C05475=1142.030,341.719,-79.384,-176.572,9.195,148.861
C05476=1142.034,341.471,-79.350,-176.575,9.190,148.861
C05477=1142.038,341.224,-79.316,-176.577,9.187,148.861
C05478=1142.042,340.976,-79.282,-176.580,9.183,148.861
C05479=1142.046,340.728,-79.248,-176.582,9.179,148.860
C05480=1142.050,340.481,-79.214,-176.585,9.175,148.860
C05481=1142.053,340.233,-79.180,-176.588,9.171,148.860
C05482=1142.058,339.985,-79.146,-176.590,9.168,148.859
C05483=1142.062,339.738,-79.112,-176.593,9.164,148.859
C05484=1142.066,339.457,-79.073,-176.595,9.160,148.859
C05485=1142.071,339.176,-79.035,-176.598,9.155,148.858
C05486=1142.075,338.896,-78.997,-176.601,9.150,148.858
C05487=1142.080,338.615,-78.959,-176.604,9.146,148.858
C05488=1142.084,338.368,-78.925,-176.606,9.143,148.857
C05489=1142.088,338.120,-78.891,-176.609,9.139,148.857
C05490=1142.092,337.872,-78.857,-176.612,9.134,148.857
C05491=1142.096,337.625,-78.824,-176.614,9.131,148.857
C05492=1142.100,337.377,-78.790,-176.617,9.127,148.856
C05493=1142.105,337.130,-78.756,-176.619,9.124,148.856
C05494=1142.108,336.881,-78.722,-176.622,9.119,148.856
C05495=1142.112,336.634,-78.689,-176.624,9.116,148.855
C05496=1142.116,336.386,-78.655,-176.627,9.112,148.855
C05497=1142.120,336.139,-78.622,-176.630,9.108,148.855
C05498=1142.124,335.892,-78.588,-176.632,9.104,148.855
C05499=1142.128,335.643,-78.554,-176.635,9.100,148.854
C05500=1142.132,335.395,-78.521,-176.637,9.097,148.854
C05501=1142.136,335.148,-78.487,-176.640,9.093,148.854
C05502=1142.140,334.900,-78.454,-176.642,9.089,148.854
C05503=1142.145,334.653,-78.421,-176.645,9.085,148.853
C05504=1142.148,334.405,-78.387,-176.647,9.082,148.853
C05505=1142.152,334.157,-78.354,-176.650,9.078,148.853
C05506=1142.156,333.909,-78.320,-176.653,9.074,148.853
C05507=1142.161,333.661,-78.287,-176.655,9.070,148.852
C05508=1142.165,333.414,-78.253,-176.658,9.066,148.852
C05509=1142.169,333.166,-78.220,-176.660,9.063,148.852
C05510=1142.172,332.918,-78.186,-176.663,9.059,148.851
C05511=1142.177,332.670,-78.153,-176.666,9.055,148.851
C05512=1142.181,332.422,-78.120,-176.668,9.051,148.851
C05513=1142.185,332.175,-78.086,-176.670,9.048,148.851
C05514=1142.189,331.928,-78.053,-176.673,9.044,148.850
C05515=1142.193,331.680,-78.020,-176.676,9.040,148.850
C05516=1142.197,331.432,-77.986,-176.679,9.036,148.850
C05517=1142.201,331.184,-77.953,-176.681,9.032,148.850
C05518=1142.205,330.936,-77.920,-176.683,9.029,148.849
C05519=1142.209,330.688,-77.887,-176.686,9.025,148.849
C05520=1142.213,330.441,-77.853,-176.689,9.021,148.849
C05521=1142.217,330.193,-77.820,-176.692,9.017,148.849
C05522=1142.221,329.945,-77.787,-176.694,9.014,148.848
C05523=1142.225,329.697,-77.754,-176.697,9.010,148.848
C05524=1142.229,329.450,-77.721,-176.699,9.006,148.848
C05525=1142.234,329.202,-77.688,-176.702,9.002,148.848
C05526=1142.237,328.954,-77.655,-176.704,8.999,148.847
C05527=1142.241,328.707,-77.622,-176.707,8.995,148.847
C05528=1142.245,328.459,-77.589,-176.709,8.992,148.847
C05529=1142.249,328.211,-77.556,-176.712,8.988,148.847
C05530=1142.254,327.964,-77.522,-176.715,8.984,148.847
C05531=1142.258,327.716,-77.489,-176.717,8.980,148.846
C05532=1142.262,327.468,-77.456,-176.719,8.977,148.846
C05533=1142.266,327.220,-77.424,-176.722,8.973,148.846
C05534=1142.270,326.972,-77.391,-176.725,8.969,148.846
C05535=1142.274,326.725,-77.358,-176.728,8.965,148.845
C05536=1142.278,326.477,-77.325,-176.730,8.962,148.845
C05537=1142.282,326.229,-77.292,-176.733,8.958,148.845
C05538=1142.286,325.981,-77.259,-176.735,8.955,148.845
C05539=1142.291,325.733,-77.226,-176.738,8.951,148.844
C05540=1142.294,325.486,-77.194,-176.740,8.947,148.844
C05541=1142.298,325.238,-77.160,-176.743,8.943,148.844
C05542=1142.302,324.990,-77.127,-176.745,8.940,148.844
C05543=1142.307,324.742,-77.095,-176.748,8.936,148.843
C05544=1142.310,324.494,-77.062,-176.750,8.932,148.843
C05545=1142.314,324.247,-77.029,-176.753,8.928,148.843
C05546=1142.319,323.998,-76.997,-176.756,8.925,148.843
C05547=1142.323,323.751,-76.963,-176.759,8.921,148.843
C05548=1142.326,323.503,-76.931,-176.761,8.918,148.842
C05549=1142.331,323.255,-76.898,-176.764,8.914,148.842
C05550=1142.335,323.007,-76.865,-176.766,8.910,148.842
C05551=1142.339,322.759,-76.833,-176.769,8.906,148.842
C05552=1142.343,322.511,-76.800,-176.771,8.903,148.842
C05553=1142.347,322.264,-76.767,-176.774,8.899,148.841
C05554=1142.351,322.016,-76.735,-176.777,8.896,148.841
C05555=1142.355,321.768,-76.702,-176.780,8.892,148.841
C05556=1142.360,321.520,-76.670,-176.782,8.888,148.841
C05557=1142.363,321.273,-76.637,-176.785,8.884,148.840
C05558=1142.368,321.024,-76.605,-176.787,8.881,148.840
C05559=1142.371,320.777,-76.572,-176.790,8.877,148.840
C05560=1142.375,320.529,-76.540,-176.793,8.874,148.840
C05561=1142.380,320.281,-76.507,-176.795,8.870,148.840
C05562=1142.383,320.033,-76.475,-176.798,8.866,148.839
C05563=1142.388,319.785,-76.443,-176.800,8.863,148.839
C05564=1142.392,319.538,-76.410,-176.803,8.859,148.839
C05565=1142.396,319.289,-76.378,-176.805,8.856,148.839
C05566=1142.400,319.042,-76.345,-176.808,8.852,148.839
C05567=1142.404,318.794,-76.313,-176.811,8.848,148.838
C05568=1142.408,318.546,-76.281,-176.814,8.844,148.838
C05569=1142.412,318.298,-76.248,-176.816,8.841,148.838
C05570=1142.416,318.051,-76.216,-176.819,8.837,148.838
C05571=1142.421,317.802,-76.184,-176.821,8.834,148.838
C05572=1142.424,317.555,-76.151,-176.823,8.830,148.837
C05573=1142.428,317.306,-76.119,-176.826,8.826,148.837
C05574=1142.432,317.058,-76.087,-176.829,8.823,148.837
C05575=1142.437,316.811,-76.055,-176.832,8.819,148.837
C05576=1142.441,316.563,-76.023,-176.834,8.816,148.837
C05577=1142.445,316.315,-75.990,-176.837,8.812,148.836
C05578=1142.449,316.067,-75.958,-176.839,8.808,148.836
C05579=1142.453,315.819,-75.926,-176.843,8.805,148.836
C05580=1142.458,315.571,-75.894,-176.845,8.801,148.836
C05581=1142.461,315.323,-75.863,-176.847,8.798,148.836
C05582=1142.465,315.076,-75.829,-176.850,8.794,148.836
C05583=1142.469,314.828,-75.798,-176.853,8.791,148.835
C05584=1142.474,314.580,-75.765,-176.855,8.787,148.835
C05585=1142.478,314.332,-75.734,-176.858,8.783,148.835
C05586=1142.482,314.084,-75.702,-176.860,8.780,148.835
C05587=1142.486,313.835,-75.669,-176.863,8.776,148.835
C05588=1142.490,313.558,-75.634,-176.866,8.772,148.834
C05589=1142.495,313.280,-75.598,-176.869,8.768,148.834
C05590=1142.500,313.003,-75.562,-176.872,8.764,148.834
C05591=1142.504,312.725,-75.526,-176.875,8.760,148.834
C05592=1142.508,312.477,-75.494,-176.878,8.757,148.834
C05593=1142.513,312.229,-75.462,-176.880,8.754,148.833
C05594=1142.516,311.981,-75.431,-176.883,8.750,148.833
C05595=1142.521,311.732,-75.399,-176.885,8.746,148.833
C05596=1142.526,311.485,-75.367,-176.888,8.743,148.833
C05597=1142.529,311.237,-75.335,-176.891,8.739,148.833
C05598=1142.533,310.989,-75.304,-176.893,8.736,148.833
C05599=1142.538,310.741,-75.272,-176.896,8.732,148.832
C05600=1142.542,310.493,-75.240,-176.898,8.729,148.832
C05601=1142.545,310.245,-75.208,-176.901,8.725,148.832
C05602=1142.550,309.998,-75.176,-176.904,8.722,148.832
C05603=1142.553,309.750,-75.145,-176.906,8.718,148.832
C05604=1142.559,309.502,-75.113,-176.909,8.714,148.832
C05605=1142.562,309.253,-75.081,-176.912,8.711,148.832
C05606=1142.566,309.005,-75.049,-176.915,8.707,148.831
C05607=1142.570,308.758,-75.018,-176.917,8.704,148.831
C05608=1142.574,308.509,-74.987,-176.920,8.701,148.831
C05609=1142.580,308.262,-74.955,-176.923,8.697,148.831
C05610=1142.583,308.014,-74.923,-176.925,8.693,148.831
C05611=1142.587,307.766,-74.891,-176.927,8.690,148.831
C05612=1142.592,307.518,-74.860,-176.930,8.686,148.830
C05613=1142.595,307.270,-74.829,-176.933,8.683,148.830
C05614=1142.600,307.022,-74.797,-176.936,8.679,148.830
C05615=1142.604,306.774,-74.766,-176.938,8.676,148.830
C05616=1142.608,306.526,-74.734,-176.941,8.673,148.830
C05617=1142.612,306.278,-74.702,-176.944,8.669,148.830
C05618=1142.617,306.030,-74.671,-176.946,8.666,148.830
C05619=1142.621,305.782,-74.639,-176.949,8.662,148.829
C05620=1142.625,305.533,-74.608,-176.952,8.658,148.829
C05621=1142.629,305.286,-74.577,-176.954,8.655,148.829
C05622=1142.633,305.038,-74.545,-176.957,8.651,148.829
C05623=1142.637,304.790,-74.514,-176.960,8.648,148.829
C05624=1142.641,304.542,-74.482,-176.962,8.645,148.829
C05625=1142.646,304.294,-74.452,-176.965,8.641,148.829
C05626=1142.649,304.046,-74.420,-176.968,8.638,148.829
C05627=1142.654,303.798,-74.389,-176.970,8.634,148.828
C05628=1142.658,303.550,-74.357,-176.973,8.630,148.828
C05629=1142.662,303.302,-74.326,-176.976,8.627,148.828
C05630=1142.667,303.054,-74.296,-176.978,8.624,148.828
C05631=1142.671,302.806,-74.264,-176.981,8.620,148.828
C05632=1142.675,302.558,-74.233,-176.983,8.617,148.828
C05633=1142.679,302.310,-74.201,-176.986,8.614,148.828
C05634=1142.683,302.062,-74.170,-176.989,8.610,148.827
C05635=1142.688,301.813,-74.139,-176.991,8.606,148.827
C05636=1142.692,301.566,-74.108,-176.994,8.604,148.827
C05637=1142.696,301.317,-74.077,-176.997,8.599,148.827
C05638=1142.700,301.070,-74.046,-176.999,8.596,148.827
C05639=1142.704,300.822,-74.015,-177.002,8.593,148.827
C05640=1142.708,300.574,-73.984,-177.005,8.589,148.827
C05641=1142.713,300.326,-73.953,-177.007,8.586,148.827
C05642=1142.716,300.078,-73.921,-177.010,8.583,148.827
C05643=1142.721,299.830,-73.890,-177.013,8.579,148.826
C05644=1142.725,299.581,-73.859,-177.015,8.576,148.826
C05645=1142.729,299.334,-73.829,-177.018,8.573,148.826
C05646=1142.733,299.086,-73.798,-177.021,8.569,148.826
C05647=1142.737,298.838,-73.767,-177.023,8.565,148.826
C05648=1142.742,298.590,-73.736,-177.026,8.562,148.826
C05649=1142.746,298.342,-73.705,-177.029,8.559,148.826
C05650=1142.750,298.093,-73.674,-177.031,8.555,148.825
C05651=1142.754,297.845,-73.644,-177.034,8.552,148.825
C05652=1142.758,297.597,-73.613,-177.037,8.549,148.825
C05653=1142.763,297.349,-73.581,-177.039,8.545,148.825
C05654=1142.767,297.101,-73.550,-177.042,8.542,148.825
C05655=1142.770,296.853,-73.520,-177.045,8.539,148.825
C05656=1142.775,296.605,-73.489,-177.048,8.535,148.825
C05657=1142.780,296.357,-73.458,-177.050,8.532,148.825
C05658=1142.783,296.109,-73.428,-177.053,8.528,148.825
C05659=1142.788,295.861,-73.397,-177.056,8.525,148.825
C05660=1142.792,295.613,-73.366,-177.058,8.521,148.824
C05661=1142.795,295.364,-73.336,-177.061,8.518,148.824
C05662=1142.800,295.117,-73.305,-177.063,8.515,148.824
C05663=1142.805,294.869,-73.274,-177.066,8.511,148.824
C05664=1142.809,294.621,-73.244,-177.069,8.508,148.824
C05665=1142.813,294.372,-73.213,-177.071,8.505,148.824
C05666=1142.817,294.124,-73.182,-177.074,8.501,148.824
C05667=1142.821,293.877,-73.152,-177.077,8.498,148.824
C05668=1142.825,293.628,-73.121,-177.080,8.495,148.824
C05669=1142.830,293.379,-73.091,-177.082,8.492,148.824
C05670=1142.834,293.132,-73.061,-177.085,8.488,148.823
C05671=1142.839,292.884,-73.030,-177.088,8.485,148.823
C05672=1142.842,292.635,-72.999,-177.090,8.481,148.823
C05673=1142.846,292.388,-72.969,-177.093,8.478,148.823
C05674=1142.850,292.140,-72.938,-177.096,8.474,148.823
C05675=1142.855,291.891,-72.908,-177.098,8.471,148.823
C05676=1142.858,291.643,-72.878,-177.101,8.468,148.823
C05677=1142.863,291.395,-72.847,-177.104,8.464,148.823
C05678=1142.868,291.147,-72.816,-177.107,8.461,148.823
C05679=1142.872,290.899,-72.786,-177.109,8.458,148.823
C05680=1142.876,290.651,-72.756,-177.112,8.455,148.823
C05681=1142.880,290.402,-72.725,-177.115,8.451,148.823
C05682=1142.884,290.154,-72.695,-177.118,8.448,148.823
C05683=1142.889,289.906,-72.665,-177.120,8.445,148.822
C05684=1142.893,289.658,-72.634,-177.123,8.442,148.822
C05685=1142.897,289.411,-72.604,-177.126,8.438,148.822
C05686=1142.901,289.162,-72.575,-177.128,8.434,148.822
C05687=1142.905,288.914,-72.544,-177.131,8.432,148.822
C05688=1142.909,288.666,-72.514,-177.133,8.428,148.822
C05689=1142.914,288.417,-72.484,-177.136,8.425,148.822
C05690=1142.918,288.170,-72.453,-177.139,8.421,148.822
C05691=1142.923,287.921,-72.423,-177.142,8.418,148.822
C05692=1142.927,287.646,-72.390,-177.145,8.415,148.822
C05693=1142.932,287.371,-72.356,-177.148,8.410,148.822
C05694=1142.937,287.095,-72.323,-177.151,8.408,148.822
C05695=1142.941,286.820,-72.289,-177.154,8.403,148.821
C05696=1142.945,286.572,-72.260,-177.156,8.401,148.822
C05697=1142.949,286.323,-72.229,-177.159,8.397,148.821
C05698=1142.954,286.075,-72.199,-177.162,8.394,148.821
C05699=1142.957,285.827,-72.169,-177.164,8.390,148.821
C05700=1142.962,285.578,-72.139,-177.167,8.387,148.821
C05701=1142.966,285.331,-72.109,-177.170,8.384,148.821
C05702=1142.970,285.082,-72.080,-177.173,8.380,148.821
C05703=1142.975,284.834,-72.050,-177.175,8.377,148.821
C05704=1142.979,284.586,-72.019,-177.178,8.374,148.821
C05705=1142.983,284.338,-71.990,-177.181,8.371,148.821
C05706=1142.987,284.090,-71.960,-177.183,8.368,148.821
C05707=1142.992,283.842,-71.930,-177.186,8.364,148.821
C05708=1142.996,283.594,-71.900,-177.189,8.361,148.821
C05709=1143.001,283.345,-71.871,-177.192,8.358,148.821
C05710=1143.004,283.098,-71.841,-177.194,8.355,148.821
C05711=1143.009,282.849,-71.811,-177.197,8.352,148.821
C05712=1143.014,282.601,-71.781,-177.200,8.348,148.821
C05713=1143.017,282.353,-71.751,-177.202,8.345,148.820
C05714=1143.022,282.105,-71.721,-177.205,8.342,148.821
C05715=1143.027,281.856,-71.691,-177.208,8.339,148.820
C05716=1143.031,281.608,-71.662,-177.210,8.336,148.820
C05717=1143.035,281.360,-71.633,-177.213,8.332,148.820
C05718=1143.039,281.112,-71.602,-177.216,8.329,148.820
C05719=1143.043,280.864,-71.573,-177.219,8.326,148.820
C05720=1143.047,280.616,-71.543,-177.221,8.322,148.820
C05721=1143.052,280.367,-71.513,-177.224,8.320,148.820
C05722=1143.056,280.119,-71.484,-177.227,8.315,148.820
C05723=1143.060,279.870,-71.454,-177.230,8.313,148.820
C05724=1143.065,279.622,-71.425,-177.232,8.310,148.820
C05725=1143.068,279.375,-71.395,-177.235,8.306,148.820
C05726=1143.073,279.126,-71.365,-177.238,8.303,148.820
C05727=1143.077,278.878,-71.336,-177.241,8.300,148.820
C05728=1143.081,278.630,-71.306,-177.243,8.296,148.820
C05729=1143.085,278.381,-71.277,-177.246,8.293,148.820
C05730=1143.089,278.133,-71.248,-177.248,8.290,148.820
C05731=1143.094,277.885,-71.218,-177.251,8.287,148.820
C05732=1143.098,277.637,-71.189,-177.254,8.284,148.820
C05733=1143.102,277.388,-71.159,-177.257,8.280,148.820
C05734=1143.106,277.140,-71.130,-177.260,8.277,148.820
C05735=1143.111,276.893,-71.101,-177.262,8.274,148.820
C05736=1143.115,276.644,-71.071,-177.265,8.271,148.820
C05737=1143.119,276.396,-71.042,-177.268,8.268,148.820
C05738=1143.124,276.147,-71.013,-177.271,8.264,148.820
C05739=1143.128,275.899,-70.984,-177.273,8.261,148.819
C05740=1143.132,275.651,-70.954,-177.276,8.258,148.820
C05741=1143.136,275.402,-70.925,-177.279,8.255,148.820
C05742=1143.140,275.154,-70.895,-177.281,8.252,148.819
C05743=1143.145,274.906,-70.866,-177.284,8.249,148.819
C05744=1143.149,274.658,-70.837,-177.287,8.246,148.820
C05745=1143.154,274.409,-70.808,-177.290,8.242,148.819
C05746=1143.158,274.161,-70.778,-177.292,8.239,148.819
C05747=1143.162,273.913,-70.749,-177.295,8.236,148.819
C05748=1143.166,273.665,-70.720,-177.298,8.233,148.819
C05749=1143.171,273.416,-70.691,-177.300,8.230,148.819
C05750=1143.176,273.168,-70.662,-177.303,8.227,148.819
C05751=1143.179,272.920,-70.633,-177.306,8.223,148.819
C05752=1143.183,272.672,-70.603,-177.309,8.220,148.819
C05753=1143.188,272.423,-70.575,-177.312,8.217,148.819
C05754=1143.192,272.175,-70.545,-177.314,8.214,148.819
C05755=1143.197,271.927,-70.516,-177.317,8.211,148.819
C05756=1143.201,271.678,-70.487,-177.319,8.208,148.819
C05757=1143.205,271.430,-70.459,-177.322,8.205,148.819
C05758=1143.209,271.182,-70.429,-177.325,8.202,148.819
C05759=1143.214,270.934,-70.401,-177.328,8.198,148.819
C05760=1143.218,270.686,-70.371,-177.331,8.195,148.819
C05761=1143.223,270.437,-70.343,-177.334,8.192,148.819
C05762=1143.226,270.189,-70.314,-177.336,8.189,148.819
C05763=1143.231,269.941,-70.285,-177.339,8.186,148.819
C05764=1143.235,269.692,-70.256,-177.341,8.183,148.819
C05765=1143.240,269.444,-70.226,-177.344,8.180,148.819
C05766=1143.243,269.195,-70.198,-177.347,8.177,148.819
C05767=1143.248,268.948,-70.169,-177.350,8.173,148.819
C05768=1143.253,268.699,-70.140,-177.353,8.170,148.819
C05769=1143.257,268.451,-70.111,-177.355,8.167,148.819
C05770=1143.261,268.203,-70.083,-177.358,8.164,148.819
C05771=1143.266,267.954,-70.054,-177.361,8.161,148.819
C05772=1143.270,267.706,-70.025,-177.363,8.158,148.819
C05773=1143.274,267.457,-69.997,-177.366,8.155,148.819
C05774=1143.278,267.210,-69.968,-177.369,8.152,148.819
C05775=1143.283,266.961,-69.939,-177.372,8.148,148.819
C05776=1143.287,266.712,-69.911,-177.375,8.145,148.819
C05777=1143.291,266.464,-69.882,-177.377,8.143,148.819
C05778=1143.296,266.216,-69.853,-177.380,8.139,148.819
C05779=1143.299,265.968,-69.824,-177.383,8.136,148.819
C05780=1143.304,265.719,-69.796,-177.385,8.133,148.819
C05781=1143.308,265.471,-69.768,-177.388,8.130,148.819
C05782=1143.313,265.223,-69.739,-177.390,8.127,148.819
C05783=1143.317,264.974,-69.710,-177.393,8.124,148.819
C05784=1143.321,264.726,-69.682,-177.396,8.121,148.819
C05785=1143.326,264.478,-69.653,-177.399,8.118,148.819
C05786=1143.330,264.229,-69.625,-177.402,8.115,148.819
C05787=1143.335,263.982,-69.596,-177.405,8.111,148.819
C05788=1143.339,263.733,-69.568,-177.407,8.109,148.819
C05789=1143.343,263.484,-69.539,-177.410,8.106,148.819
C05790=1143.347,263.236,-69.511,-177.413,8.103,148.819
C05791=1143.352,262.987,-69.483,-177.416,8.100,148.819
C05792=1143.357,262.740,-69.454,-177.418,8.096,148.819
C05793=1143.360,262.491,-69.426,-177.421,8.094,148.819
C05794=1143.364,262.243,-69.397,-177.424,8.091,148.819
C05795=1143.369,261.994,-69.369,-177.426,8.088,148.819
C05796=1143.374,261.721,-69.338,-177.430,8.084,148.820
C05797=1143.379,261.447,-69.307,-177.433,8.081,148.820
C05798=1143.383,261.174,-69.275,-177.436,8.077,148.820
C05799=1143.388,260.900,-69.244,-177.439,8.074,148.820
C05800=1143.392,260.652,-69.216,-177.441,8.071,148.820
C05801=1143.397,260.404,-69.188,-177.444,8.068,148.820
C05802=1143.401,260.155,-69.159,-177.447,8.065,148.820
C05803=1143.405,259.907,-69.132,-177.449,8.062,148.820
C05804=1143.410,259.658,-69.103,-177.453,8.059,148.820
C05805=1143.414,259.410,-69.075,-177.456,8.056,148.820
C05806=1143.418,259.162,-69.047,-177.458,8.053,148.820
C05807=1143.423,258.914,-69.019,-177.461,8.049,148.820
C05808=1143.427,258.665,-68.990,-177.463,8.047,148.820
C05809=1143.431,258.417,-68.963,-177.466,8.044,148.820
C05810=1143.436,258.168,-68.934,-177.469,8.041,148.820
C05811=1143.440,257.920,-68.907,-177.472,8.038,148.820
C05812=1143.444,257.671,-68.879,-177.475,8.035,148.820
C05813=1143.449,257.423,-68.850,-177.477,8.032,148.820
C05814=1143.453,257.174,-68.822,-177.480,8.029,148.820
C05815=1143.457,256.927,-68.794,-177.483,8.026,148.820
C05816=1143.462,256.678,-68.766,-177.485,8.023,148.820
C05817=1143.466,256.429,-68.739,-177.488,8.020,148.820
C05818=1143.471,256.181,-68.711,-177.491,8.017,148.820
C05819=1143.474,255.933,-68.683,-177.494,8.014,148.820
C05820=1143.480,255.685,-68.654,-177.497,8.011,148.820
C05821=1143.483,255.436,-68.626,-177.499,8.008,148.820
C05822=1143.488,255.187,-68.599,-177.502,8.005,148.820
C05823=1143.492,254.940,-68.571,-177.504,8.002,148.820
C05824=1143.497,254.691,-68.543,-177.507,7.999,148.820
C05825=1143.501,254.442,-68.516,-177.510,7.996,148.820
C05826=1143.505,254.194,-68.487,-177.513,7.993,148.821
C05827=1143.510,253.946,-68.460,-177.516,7.990,148.821
C05828=1143.514,253.697,-68.433,-177.518,7.987,148.821
C05829=1143.519,253.448,-68.404,-177.522,7.984,148.821
C05830=1143.523,253.200,-68.376,-177.525,7.981,148.821
C05831=1143.527,252.951,-68.349,-177.527,7.978,148.821
C05832=1143.531,252.703,-68.321,-177.530,7.975,148.821
C05833=1143.536,252.455,-68.294,-177.533,7.972,148.821
C05834=1143.540,252.206,-68.266,-177.535,7.969,148.821
C05835=1143.544,251.958,-68.238,-177.538,7.966,148.821
C05836=1143.550,251.710,-68.210,-177.541,7.963,148.821
C05837=1143.553,251.461,-68.182,-177.544,7.960,148.821
C05838=1143.558,251.213,-68.155,-177.546,7.957,148.821
C05839=1143.562,250.965,-68.127,-177.549,7.954,148.821
C05840=1143.566,250.716,-68.100,-177.552,7.951,148.821
C05841=1143.571,250.468,-68.072,-177.555,7.948,148.821
C05842=1143.575,250.219,-68.045,-177.558,7.945,148.821
C05843=1143.579,249.971,-68.017,-177.560,7.942,148.821
C05844=1143.584,249.722,-67.990,-177.563,7.939,148.822
C05845=1143.589,249.474,-67.963,-177.566,7.937,148.822
C05846=1143.593,249.226,-67.935,-177.569,7.934,148.822
C05847=1143.597,248.976,-67.907,-177.572,7.931,148.822
C05848=1143.601,248.729,-67.880,-177.574,7.928,148.822
C05849=1143.606,248.480,-67.853,-177.577,7.925,148.822
C05850=1143.610,248.231,-67.825,-177.580,7.922,148.822
C05851=1143.614,247.983,-67.797,-177.583,7.919,148.822
C05852=1143.619,247.735,-67.770,-177.585,7.917,148.822
C05853=1143.624,247.486,-67.743,-177.588,7.914,148.822
C05854=1143.627,247.237,-67.715,-177.590,7.911,148.822
C05855=1143.632,246.989,-67.688,-177.593,7.908,148.822
C05856=1143.637,246.740,-67.661,-177.596,7.905,148.822
C05857=1143.641,246.492,-67.634,-177.599,7.902,148.823
C05858=1143.646,246.244,-67.606,-177.601,7.899,148.822
C05859=1143.650,245.995,-67.579,-177.604,7.896,148.822
C05860=1143.654,245.746,-67.552,-177.607,7.893,148.823
C05861=1143.658,245.498,-67.525,-177.610,7.890,148.823
C05862=1143.663,245.250,-67.497,-177.612,7.887,148.823
C05863=1143.667,245.002,-67.470,-177.615,7.884,148.823
C05864=1143.671,244.753,-67.443,-177.618,7.882,148.823
C05865=1143.676,244.504,-67.416,-177.621,7.879,148.823
C05866=1143.681,244.256,-67.389,-177.624,7.876,148.823
C05867=1143.685,244.007,-67.362,-177.626,7.873,148.823
C05868=1143.689,243.759,-67.335,-177.630,7.870,148.823
C05869=1143.693,243.510,-67.307,-177.632,7.867,148.823
C05870=1143.698,243.262,-67.280,-177.635,7.864,148.824
C05871=1143.702,243.013,-67.253,-177.638,7.861,148.824
C05872=1143.707,242.765,-67.226,-177.641,7.858,148.824
C05873=1143.711,242.517,-67.200,-177.644,7.856,148.824
C05874=1143.716,242.268,-67.172,-177.646,7.853,148.824
C05875=1143.720,242.020,-67.145,-177.649,7.850,148.824
C05876=1143.724,241.771,-67.118,-177.652,7.847,148.824
C05877=1143.728,241.522,-67.092,-177.654,7.845,148.824
C05878=1143.733,241.274,-67.064,-177.657,7.842,148.824
C05879=1143.738,241.025,-67.037,-177.660,7.839,148.824
C05880=1143.742,240.777,-67.010,-177.662,7.836,148.824
C05881=1143.746,240.529,-66.984,-177.665,7.833,148.824
C05882=1143.751,240.280,-66.957,-177.668,7.830,148.824
C05883=1143.755,240.032,-66.930,-177.671,7.827,148.825
C05884=1143.760,239.783,-66.904,-177.674,7.824,148.825
C05885=1143.764,239.534,-66.877,-177.676,7.821,148.825
C05886=1143.769,239.286,-66.850,-177.679,7.818,148.825
C05887=1143.772,239.037,-66.823,-177.682,7.816,148.825
C05888=1143.777,238.789,-66.796,-177.685,7.813,148.825
C05889=1143.782,238.540,-66.769,-177.688,7.810,148.825
C05890=1143.786,238.292,-66.742,-177.690,7.807,148.825
C05891=1143.790,238.043,-66.716,-177.693,7.805,148.825
C05892=1143.795,237.794,-66.689,-177.695,7.802,148.825
C05893=1143.799,237.546,-66.663,-177.699,7.799,148.826
C05894=1143.804,237.298,-66.636,-177.701,7.796,148.826
C05895=1143.808,237.049,-66.610,-177.704,7.793,148.826
C05896=1143.813,236.800,-66.583,-177.707,7.790,148.826
C05897=1143.817,236.552,-66.556,-177.710,7.787,148.826
C05898=1143.821,236.304,-66.529,-177.713,7.785,148.826
C05899=1143.826,236.054,-66.503,-177.715,7.782,148.826
C05900=1143.831,235.783,-66.474,-177.718,7.779,148.826
C05901=1143.836,235.512,-66.445,-177.721,7.776,148.826
C05902=1143.840,235.239,-66.416,-177.724,7.773,148.827
C05903=1143.845,234.967,-66.387,-177.728,7.769,148.827
C05904=1143.850,234.719,-66.360,-177.730,7.767,148.827
C05905=1143.854,234.470,-66.334,-177.733,7.764,148.827
C05906=1143.858,234.222,-66.307,-177.735,7.762,148.827
C05907=1143.863,233.973,-66.281,-177.738,7.759,148.827
C05908=1143.867,233.724,-66.254,-177.741,7.756,148.827
C05909=1143.871,233.476,-66.228,-177.744,7.753,148.827
C05910=1143.876,233.227,-66.201,-177.747,7.750,148.827
C05911=1143.881,232.980,-66.175,-177.750,7.747,148.828
C05912=1143.886,232.730,-66.149,-177.753,7.744,148.828
C05913=1143.890,232.482,-66.123,-177.755,7.741,148.828
C05914=1143.895,232.233,-66.096,-177.758,7.739,148.828
C05915=1143.898,231.985,-66.070,-177.761,7.736,148.828
C05916=1143.903,231.736,-66.044,-177.763,7.734,148.828
C05917=1143.907,231.488,-66.017,-177.766,7.731,148.828
C05918=1143.912,231.239,-65.991,-177.769,7.728,148.828
C05919=1143.917,230.990,-65.965,-177.772,7.725,148.828
C05920=1143.920,230.742,-65.938,-177.775,7.722,148.829
C05921=1143.925,230.493,-65.913,-177.778,7.719,148.829
C05922=1143.930,230.245,-65.886,-177.780,7.717,148.829
C05923=1143.934,229.996,-65.860,-177.783,7.714,148.829
C05924=1143.938,229.747,-65.834,-177.786,7.711,148.829
C05925=1143.943,229.499,-65.807,-177.788,7.708,148.829
C05926=1143.947,229.250,-65.782,-177.792,7.706,148.829
C05927=1143.951,229.001,-65.756,-177.794,7.703,148.829
C05928=1143.957,228.753,-65.729,-177.797,7.701,148.829
C05929=1143.961,228.505,-65.703,-177.799,7.698,148.830
C05930=1143.965,228.256,-65.678,-177.802,7.695,148.830
C05931=1143.969,228.007,-65.652,-177.805,7.692,148.830
C05932=1143.974,227.758,-65.625,-177.808,7.690,148.830
C05933=1143.978,227.510,-65.599,-177.811,7.687,148.830
C05934=1143.983,227.262,-65.574,-177.814,7.684,148.830
C05935=1143.987,227.013,-65.548,-177.816,7.682,148.830
C05936=1143.992,226.764,-65.521,-177.819,7.679,148.830
C05937=1143.996,226.515,-65.495,-177.822,7.676,148.831
C05938=1144.000,226.267,-65.469,-177.825,7.673,148.831
C05939=1144.005,226.019,-65.444,-177.828,7.670,148.831
C05940=1144.010,225.769,-65.418,-177.831,7.667,148.831
C05941=1144.014,225.521,-65.392,-177.833,7.665,148.831
C05942=1144.019,225.272,-65.366,-177.836,7.662,148.831
C05943=1144.023,225.024,-65.340,-177.839,7.660,148.832
C05944=1144.027,224.776,-65.314,-177.842,7.657,148.832
C05945=1144.032,224.527,-65.289,-177.844,7.654,148.832
C05946=1144.037,224.278,-65.262,-177.847,7.652,148.832
C05947=1144.041,224.030,-65.237,-177.849,7.649,148.832
C05948=1144.046,223.781,-65.211,-177.853,7.646,148.832
C05949=1144.050,223.532,-65.185,-177.855,7.643,148.832
C05950=1144.054,223.283,-65.160,-177.858,7.641,148.832
C05951=1144.059,223.035,-65.134,-177.860,7.638,148.833
C05952=1144.063,222.786,-65.108,-177.863,7.636,148.833
C05953=1144.067,222.537,-65.083,-177.867,7.633,148.833
C05954=1144.072,222.289,-65.057,-177.869,7.630,148.833
C05955=1144.076,222.040,-65.032,-177.872,7.627,148.833
C05956=1144.081,221.791,-65.005,-177.874,7.625,148.833
C05957=1144.086,221.543,-64.980,-177.877,7.622,148.833
C05958=1144.090,221.294,-64.954,-177.880,7.620,148.834
C05959=1144.095,221.045,-64.929,-177.883,7.617,148.834
C05960=1144.100,220.797,-64.904,-177.886,7.614,148.834
C05961=1144.104,220.548,-64.878,-177.888,7.612,148.834
C05962=1144.108,220.299,-64.852,-177.891,7.609,148.834
C05963=1144.113,220.051,-64.827,-177.894,7.606,148.834
C05964=1144.117,219.802,-64.801,-177.897,7.603,148.834
C05965=1144.122,219.554,-64.775,-177.900,7.600,148.835
C05966=1144.127,219.305,-64.751,-177.903,7.599,148.835
C05967=1144.131,219.056,-64.725,-177.905,7.596,148.835
C05968=1144.135,218.807,-64.699,-177.908,7.593,148.835
C05969=1144.139,218.560,-64.674,-177.911,7.590,148.835
C05970=1144.143,218.311,-64.649,-177.914,7.588,148.835
C05971=1144.149,218.062,-64.624,-177.916,7.585,148.836
C05972=1144.153,217.813,-64.598,-177.919,7.582,148.836
C05973=1144.157,217.564,-64.572,-177.922,7.579,148.836
C05974=1144.162,217.316,-64.548,-177.925,7.578,148.836
C05975=1144.166,217.067,-64.522,-177.927,7.575,148.836
C05976=1144.171,216.819,-64.497,-177.930,7.572,148.836
C05977=1144.176,216.569,-64.472,-177.933,7.569,148.836
C05978=1144.180,216.320,-64.446,-177.936,7.566,148.837
C05979=1144.184,216.073,-64.421,-177.939,7.564,148.837
C05980=1144.189,215.823,-64.396,-177.941,7.561,148.837
C05981=1144.193,215.575,-64.371,-177.945,7.559,148.837
C05982=1144.198,215.326,-64.345,-177.947,7.556,148.837
C05983=1144.203,215.078,-64.320,-177.950,7.554,148.837
C05984=1144.207,214.829,-64.294,-177.952,7.551,148.838
C05985=1144.211,214.580,-64.270,-177.956,7.548,148.838
C05986=1144.216,214.332,-64.245,-177.958,7.546,148.838
C05987=1144.220,214.082,-64.220,-177.961,7.543,148.838
C05988=1144.225,213.834,-64.194,-177.964,7.541,148.838
C05989=1144.229,213.585,-64.169,-177.967,7.538,148.839
C05990=1144.234,213.337,-64.144,-177.969,7.536,148.839
C05991=1144.238,213.087,-64.119,-177.972,7.533,148.839
C05992=1144.243,212.839,-64.094,-177.975,7.530,148.839
C05993=1144.247,212.590,-64.069,-177.978,7.527,148.839
C05994=1144.252,212.342,-64.044,-177.980,7.525,148.839
C05995=1144.256,212.093,-64.019,-177.983,7.523,148.840
C05996=1144.261,211.845,-63.994,-177.986,7.520,148.840
C05997=1144.265,211.596,-63.970,-177.988,7.518,148.840
C05998=1144.270,211.347,-63.945,-177.992,7.515,148.840
C05999=1144.275,211.099,-63.919,-177.994,7.512,148.840
C06000=1144.278,210.850,-63.895,-177.997,7.509,148.840
C06001=1144.284,210.601,-63.870,-178.000,7.507,148.841
C06002=1144.288,210.352,-63.844,-178.003,7.505,148.841
C06003=1144.292,210.104,-63.820,-178.006,7.502,148.841
C06004=1144.297,209.832,-63.793,-178.009,7.499,148.841
C06005=1144.303,209.562,-63.766,-178.012,7.496,148.841
C06006=1144.307,209.291,-63.739,-178.015,7.494,148.842
C06007=1144.312,209.021,-63.712,-178.018,7.491,148.842
C06008=1144.317,208.772,-63.687,-178.020,7.489,148.842
C06009=1144.321,208.524,-63.662,-178.023,7.486,148.842
C06010=1144.325,208.275,-63.637,-178.026,7.483,148.842
C06011=1144.330,208.026,-63.613,-178.029,7.481,148.843
C06012=1144.335,207.777,-63.588,-178.031,7.478,148.843
C06013=1144.340,207.528,-63.563,-178.034,7.476,148.843
C06014=1144.344,207.280,-63.539,-178.038,7.473,148.843
C06015=1144.349,207.031,-63.514,-178.040,7.471,148.843
C06016=1144.353,206.782,-63.490,-178.043,7.468,148.843
C06017=1144.358,206.534,-63.465,-178.046,7.465,148.844
C06018=1144.361,206.285,-63.440,-178.048,7.463,148.844
C06019=1144.367,206.036,-63.416,-178.051,7.461,148.844
C06020=1144.371,205.787,-63.392,-178.054,7.458,148.844
C06021=1144.375,205.539,-63.366,-178.056,7.456,148.844
C06022=1144.380,205.290,-63.342,-178.060,7.453,148.845
C06023=1144.385,205.041,-63.317,-178.062,7.450,148.845
C06024=1144.389,204.793,-63.293,-178.065,7.449,148.845
C06025=1144.394,204.544,-63.268,-178.068,7.446,148.845
C06026=1144.398,204.295,-63.244,-178.071,7.443,148.845
C06027=1144.403,204.046,-63.219,-178.073,7.441,148.846
C06028=1144.407,203.797,-63.195,-178.076,7.438,148.846
C06029=1144.412,203.549,-63.170,-178.079,7.435,148.846
C06030=1144.417,203.300,-63.146,-178.082,7.433,148.846
C06031=1144.420,203.051,-63.122,-178.084,7.430,148.846
C06032=1144.425,202.802,-63.097,-178.088,7.428,148.847
C06033=1144.430,202.554,-63.073,-178.090,7.426,148.847
C06034=1144.435,202.305,-63.048,-178.093,7.423,148.847
C06035=1144.439,202.056,-63.025,-178.095,7.421,148.847
C06036=1144.443,201.807,-63.001,-178.098,7.418,148.847
C06037=1144.449,201.558,-62.976,-178.102,7.416,148.848
C06038=1144.452,201.309,-62.951,-178.104,7.414,148.848
C06039=1144.457,201.061,-62.927,-178.107,7.411,148.848
C06040=1144.462,200.812,-62.903,-178.110,7.408,148.848
C06041=1144.466,200.564,-62.879,-178.113,7.406,148.849
C06042=1144.471,200.315,-62.855,-178.115,7.404,148.849
C06043=1144.476,200.065,-62.830,-178.118,7.401,148.849
C06044=1144.480,199.817,-62.806,-178.121,7.399,148.849
C06045=1144.484,199.568,-62.782,-178.124,7.396,148.849
C06046=1144.489,199.320,-62.757,-178.126,7.394,148.850
C06047=1144.494,199.070,-62.734,-178.129,7.391,148.850
C06048=1144.498,198.822,-62.710,-178.132,7.389,148.850
C06049=1144.502,198.573,-62.685,-178.135,7.387,148.850
C06050=1144.507,198.324,-62.661,-178.138,7.384,148.851
C06051=1144.512,198.075,-62.637,-178.140,7.382,148.851
C06052=1144.517,197.827,-62.613,-178.143,7.379,148.851
C06053=1144.520,197.578,-62.589,-178.146,7.377,148.851
C06054=1144.526,197.329,-62.565,-178.148,7.374,148.851
C06055=1144.530,197.080,-62.541,-178.152,7.372,148.852
C06056=1144.535,196.832,-62.517,-178.154,7.370,148.852
C06057=1144.539,196.583,-62.493,-178.157,7.367,148.852
C06058=1144.544,196.334,-62.469,-178.160,7.364,148.852
C06059=1144.548,196.085,-62.444,-178.163,7.363,148.853
C06060=1144.553,195.836,-62.421,-178.165,7.360,148.853
C06061=1144.557,195.587,-62.397,-178.168,7.358,148.853
C06062=1144.562,195.338,-62.374,-178.171,7.355,148.853
C06063=1144.566,195.090,-62.350,-178.174,7.353,148.853
C06064=1144.571,194.841,-62.326,-178.176,7.350,148.854
C06065=1144.576,194.592,-62.301,-178.180,7.348,148.854
C06066=1144.581,194.343,-62.278,-178.182,7.346,148.854
C06067=1144.585,194.095,-62.254,-178.185,7.343,148.854
C06068=1144.589,193.845,-62.230,-178.187,7.341,148.855
C06069=1144.594,193.597,-62.206,-178.191,7.339,148.855
C06070=1144.599,193.348,-62.183,-178.194,7.336,148.855
C06071=1144.603,193.099,-62.159,-178.196,7.334,148.855
C06072=1144.608,192.850,-62.135,-178.199,7.331,148.855
C06073=1144.612,192.602,-62.111,-178.202,7.329,148.856
C06074=1144.617,192.353,-62.088,-178.205,7.326,148.856
C06075=1144.621,192.104,-62.064,-178.207,7.325,148.856
C06076=1144.626,191.855,-62.041,-178.210,7.322,148.856
C06077=1144.631,191.606,-62.017,-178.213,7.319,148.857
C06078=1144.636,191.357,-61.993,-178.216,7.317,148.857
C06079=1144.640,191.108,-61.969,-178.219,7.315,148.857
C06080=1144.645,190.859,-61.946,-178.221,7.312,148.857
C06081=1144.649,190.611,-61.922,-178.224,7.310,148.858
C06082=1144.654,190.362,-61.898,-178.227,7.308,148.858
C06083=1144.659,190.113,-61.875,-178.230,7.305,148.858
C06084=1144.663,189.865,-61.851,-178.233,7.304,148.858
C06085=1144.668,189.616,-61.828,-178.235,7.301,148.859
C06086=1144.672,189.367,-61.805,-178.238,7.299,148.859
C06087=1144.677,189.118,-61.781,-178.241,7.296,148.859
C06088=1144.681,188.869,-61.757,-178.244,7.293,148.859
C06089=1144.686,188.620,-61.734,-178.246,7.291,148.860
C06090=1144.690,188.371,-61.711,-178.250,7.289,148.860
C06091=1144.695,188.122,-61.687,-178.252,7.287,148.860
C06092=1144.699,187.874,-61.663,-178.255,7.284,148.860
C06093=1144.704,187.625,-61.640,-178.258,7.282,148.861
C06094=1144.709,187.376,-61.617,-178.261,7.280,148.861
C06095=1144.714,187.127,-61.593,-178.263,7.278,148.861
C06096=1144.718,186.878,-61.570,-178.266,7.275,148.861
C06097=1144.723,186.629,-61.546,-178.269,7.273,148.862
C06098=1144.727,186.380,-61.524,-178.272,7.270,148.862
C06099=1144.731,186.132,-61.500,-178.274,7.268,148.862
C06100=1144.736,185.882,-61.476,-178.277,7.266,148.862
C06101=1144.741,185.633,-61.453,-178.280,7.264,148.863
C06102=1144.746,185.385,-61.430,-178.283,7.261,148.863
C06103=1144.751,185.136,-61.407,-178.285,7.259,148.863
C06104=1144.755,184.887,-61.384,-178.289,7.257,148.863
C06105=1144.759,184.638,-61.360,-178.291,7.255,148.864
C06106=1144.764,184.389,-61.337,-178.294,7.252,148.864
C06107=1144.769,184.140,-61.314,-178.297,7.250,148.864
C06108=1144.773,183.871,-61.289,-178.300,7.247,148.864
C06109=1144.779,183.601,-61.264,-178.303,7.245,148.865
C06110=1144.784,183.332,-61.239,-178.306,7.242,148.865
C06111=1144.789,183.062,-61.213,-178.308,7.240,148.865
C06112=1144.793,182.813,-61.191,-178.312,7.238,148.866
C06113=1144.798,182.564,-61.167,-178.314,7.236,148.866
C06114=1144.802,182.315,-61.144,-178.317,7.233,148.866
C06115=1144.807,182.066,-61.121,-178.320,7.231,148.866
C06116=1144.811,181.817,-61.099,-178.323,7.229,148.867
C06117=1144.816,181.568,-61.075,-178.325,7.227,148.867
C06118=1144.821,181.320,-61.052,-178.329,7.224,148.867
C06119=1144.825,181.071,-61.029,-178.331,7.222,148.867
C06120=1144.830,180.822,-61.006,-178.334,7.219,148.868
C06121=1144.835,180.573,-60.983,-178.337,7.218,148.868
C06122=1144.839,180.324,-60.960,-178.340,7.215,148.868
C06123=1144.844,180.075,-60.938,-178.342,7.213,148.869
C06124=1144.849,179.826,-60.914,-178.345,7.210,148.869
C06125=1144.853,179.577,-60.892,-178.348,7.208,148.869
C06126=1144.858,179.328,-60.868,-178.351,7.206,148.869
C06127=1144.862,179.079,-60.846,-178.353,7.204,148.870
C06128=1144.867,178.831,-60.823,-178.356,7.202,148.870
C06129=1144.872,178.582,-60.800,-178.359,7.200,148.870
C06130=1144.876,178.333,-60.777,-178.362,7.198,148.870
C06131=1144.881,178.083,-60.754,-178.365,7.195,148.871
C06132=1144.885,177.835,-60.732,-178.368,7.193,148.871
C06133=1144.890,177.586,-60.709,-178.370,7.190,148.871
C06134=1144.894,177.337,-60.687,-178.373,7.189,148.872
C06135=1144.899,177.088,-60.663,-178.376,7.186,148.872
C06136=1144.904,176.840,-60.640,-178.379,7.184,148.872
C06137=1144.909,176.590,-60.618,-178.382,7.181,148.872
C06138=1144.913,176.341,-60.595,-178.385,7.180,148.873
C06139=1144.917,176.092,-60.572,-178.387,7.178,148.873
C06140=1144.923,175.844,-60.550,-178.390,7.175,148.873
C06141=1144.927,175.595,-60.527,-178.393,7.173,148.874
C06142=1144.932,175.345,-60.504,-178.396,7.170,148.874
C06143=1144.936,175.097,-60.482,-178.398,7.169,148.874
C06144=1144.941,174.847,-60.459,-178.402,7.166,148.875
C06145=1144.945,174.599,-60.437,-178.404,7.164,148.875
C06146=1144.951,174.350,-60.414,-178.406,7.162,148.875
C06147=1144.955,174.101,-60.392,-178.410,7.160,148.875
C06148=1144.959,173.852,-60.369,-178.412,7.158,148.876
C06149=1144.965,173.603,-60.347,-178.415,7.155,148.876
C06150=1144.969,173.355,-60.324,-178.418,7.153,148.876
C06151=1144.974,173.105,-60.301,-178.420,7.151,148.876
C06152=1144.978,172.856,-60.279,-178.424,7.149,148.877
C06153=1144.983,172.607,-60.256,-178.426,7.147,148.877
C06154=1144.987,172.358,-60.234,-178.429,7.144,148.877
C06155=1144.992,172.110,-60.212,-178.432,7.142,148.878
C06156=1144.997,171.860,-60.189,-178.434,7.141,148.878
C06157=1145.001,171.612,-60.166,-178.437,7.138,148.878
C06158=1145.006,171.363,-60.145,-178.440,7.136,148.879
C06159=1145.011,171.113,-60.122,-178.443,7.134,148.879
C06160=1145.015,170.865,-60.099,-178.446,7.132,148.879
C06161=1145.020,170.616,-60.077,-178.448,7.130,148.879
C06162=1145.025,170.366,-60.055,-178.451,7.127,148.880
C06163=1145.029,170.118,-60.032,-178.454,7.126,148.880
C06164=1145.034,169.869,-60.010,-178.457,7.123,148.880
C06165=1145.039,169.620,-59.988,-178.460,7.121,148.881
C06166=1145.043,169.371,-59.965,-178.462,7.119,148.881
C06167=1145.047,169.122,-59.943,-178.466,7.117,148.881
C06168=1145.053,168.873,-59.921,-178.468,7.115,148.881
C06169=1145.057,168.624,-59.899,-178.471,7.112,148.882
C06170=1145.062,168.376,-59.877,-178.474,7.110,148.882
C06171=1145.067,168.126,-59.854,-178.476,7.108,148.882
C06172=1145.072,167.877,-59.832,-178.479,7.106,148.883
C06173=1145.076,167.628,-59.810,-178.482,7.104,148.883
C06174=1145.081,167.379,-59.788,-178.485,7.102,148.883
C06175=1145.085,167.130,-59.765,-178.488,7.099,148.884
C06176=1145.090,166.882,-59.743,-178.490,7.098,148.884
C06177=1145.095,166.632,-59.721,-178.493,7.096,148.884
C06178=1145.099,166.384,-59.700,-178.496,7.093,148.885
C06179=1145.104,166.134,-59.678,-178.499,7.091,148.885
C06180=1145.109,165.885,-59.655,-178.502,7.089,148.885
C06181=1145.114,165.636,-59.633,-178.505,7.087,148.886
C06182=1145.118,165.387,-59.612,-178.507,7.085,148.886
C06183=1145.123,165.138,-59.590,-178.510,7.082,148.886
C06184=1145.127,164.890,-59.567,-178.513,7.081,148.886
C06185=1145.132,164.641,-59.545,-178.515,7.079,148.887
C06186=1145.136,164.392,-59.523,-178.519,7.076,148.887
C06187=1145.141,164.142,-59.501,-178.521,7.074,148.887
C06188=1145.146,163.894,-59.479,-178.524,7.073,148.888
C06189=1145.151,163.644,-59.457,-178.527,7.070,148.888
C06190=1145.155,163.396,-59.435,-178.530,7.068,148.888
C06191=1145.160,163.146,-59.413,-178.532,7.066,148.889
C06192=1145.165,162.898,-59.392,-178.535,7.064,148.889
C06193=1145.169,162.648,-59.370,-178.538,7.062,148.889
C06194=1145.174,162.400,-59.348,-178.541,7.060,148.890
C06195=1145.178,162.151,-59.326,-178.544,7.058,148.890
C06196=1145.183,161.901,-59.305,-178.546,7.056,148.890
C06197=1145.188,161.653,-59.283,-178.549,7.054,148.891
C06198=1145.192,161.403,-59.261,-178.552,7.051,148.891
C06199=1145.197,161.155,-59.240,-178.555,7.050,148.891
C06200=1145.201,160.905,-59.217,-178.558,7.048,148.892
C06201=1145.206,160.657,-59.196,-178.560,7.045,148.892
C06202=1145.211,160.408,-59.174,-178.563,7.043,148.892
C06203=1145.215,160.159,-59.152,-178.566,7.042,148.893
C06204=1145.221,159.909,-59.131,-178.568,7.040,148.893
C06205=1145.225,159.660,-59.109,-178.571,7.037,148.893
C06206=1145.230,159.411,-59.087,-178.574,7.035,148.893
C06207=1145.235,159.163,-59.066,-178.577,7.034,148.894
C06208=1145.239,158.913,-59.044,-178.580,7.031,148.894
C06209=1145.244,158.664,-59.023,-178.583,7.029,148.895
C06210=1145.249,158.416,-59.001,-178.585,7.028,148.895
C06211=1145.253,158.166,-58.979,-178.588,7.025,148.895
C06212=1145.259,157.897,-58.956,-178.591,7.023,148.895
C06213=1145.263,157.628,-58.932,-178.594,7.020,148.896
C06214=1145.269,157.359,-58.909,-178.597,7.019,148.896
C06215=1145.273,157.090,-58.886,-178.600,7.016,148.897
C06216=1145.278,156.841,-58.864,-178.603,7.014,148.897
C06217=1145.283,156.593,-58.843,-178.606,7.013,148.897
C06218=1145.288,156.343,-58.822,-178.609,7.010,148.898
C06219=1145.293,156.094,-58.800,-178.611,7.008,148.898
C06220=1145.298,155.845,-58.779,-178.614,7.006,148.898
C06221=1145.303,155.596,-58.757,-178.617,7.005,148.899
C06222=1145.306,155.347,-58.736,-178.620,7.002,148.899
C06223=1145.311,155.098,-58.715,-178.623,7.000,148.899
C06224=1145.316,154.849,-58.693,-178.625,6.999,148.900
C06225=1145.321,154.600,-58.672,-178.628,6.996,148.900
C06226=1145.326,154.351,-58.650,-178.631,6.994,148.900
C06227=1145.330,154.102,-58.628,-178.634,6.992,148.901
C06228=1145.335,153.853,-58.608,-178.636,6.991,148.901
C06229=1145.339,153.604,-58.586,-178.640,6.988,148.901
C06230=1145.344,153.354,-58.565,-178.642,6.986,148.902
C06231=1145.349,153.106,-58.543,-178.645,6.985,148.902
C06232=1145.354,152.857,-58.523,-178.647,6.983,148.902
C06233=1145.359,152.608,-58.501,-178.650,6.980,148.903
C06234=1145.363,152.358,-58.480,-178.653,6.978,148.903
C06235=1145.368,152.110,-58.458,-178.656,6.977,148.903
C06236=1145.372,151.861,-58.438,-178.659,6.975,148.904
C06237=1145.378,151.611,-58.417,-178.662,6.972,148.904
C06238=1145.382,151.362,-58.395,-178.665,6.971,148.905
C06239=1145.387,151.113,-58.374,-178.667,6.969,148.905
C06240=1145.391,150.865,-58.353,-178.670,6.967,148.905
C06241=1145.396,150.615,-58.332,-178.673,6.964,148.905
C06242=1145.402,150.366,-58.311,-178.676,6.963,148.906
C06243=1145.406,150.118,-58.290,-178.678,6.961,148.906
C06244=1145.410,149.868,-58.268,-178.681,6.959,148.907
C06245=1145.415,149.618,-58.247,-178.684,6.958,148.907
C06246=1145.420,149.370,-58.226,-178.686,6.955,148.907
C06247=1145.425,149.121,-58.205,-178.689,6.953,148.908
C06248=1145.430,148.872,-58.184,-178.692,6.951,148.908
C06249=1145.434,148.623,-58.163,-178.695,6.950,148.908
C06250=1145.439,148.373,-58.142,-178.698,6.947,148.909
C06251=1145.444,148.124,-58.121,-178.701,6.945,148.909
C06252=1145.448,147.876,-58.100,-178.703,6.944,148.909
C06253=1145.453,147.626,-58.079,-178.706,6.942,148.910
C06254=1145.457,147.378,-58.058,-178.709,6.940,148.910
C06255=1145.463,147.128,-58.037,-178.712,6.937,148.910
C06256=1145.468,146.879,-58.016,-178.714,6.936,148.911
C06257=1145.471,146.630,-57.995,-178.717,6.934,148.911
C06258=1145.477,146.381,-57.974,-178.720,6.932,148.912
C06259=1145.481,146.132,-57.954,-178.722,6.930,148.912
C06260=1145.486,145.882,-57.933,-178.726,6.928,148.912
C06261=1145.491,145.634,-57.912,-178.728,6.926,148.913
C06262=1145.495,145.385,-57.891,-178.731,6.924,148.913
C06263=1145.500,145.136,-57.870,-178.734,6.923,148.913
C06264=1145.505,144.887,-57.849,-178.737,6.921,148.914
C06265=1145.510,144.638,-57.829,-178.739,6.918,148.914
C06266=1145.515,144.388,-57.808,-178.742,6.916,148.914
C06267=1145.519,144.140,-57.788,-178.745,6.915,148.915
C06268=1145.524,143.890,-57.767,-178.748,6.913,148.915
C06269=1145.528,143.641,-57.746,-178.750,6.911,148.916
C06270=1145.533,143.391,-57.725,-178.754,6.909,148.916
C06271=1145.538,143.142,-57.705,-178.756,6.907,148.916
C06272=1145.543,142.893,-57.684,-178.759,6.905,148.917
C06273=1145.547,142.644,-57.663,-178.762,6.904,148.917
C06274=1145.553,142.395,-57.642,-178.764,6.902,148.917
C06275=1145.557,142.146,-57.622,-178.767,6.900,148.918
C06276=1145.561,141.897,-57.602,-178.770,6.898,148.918
C06277=1145.567,141.648,-57.581,-178.773,6.896,148.919
C06278=1145.571,141.399,-57.560,-178.776,6.894,148.919
C06279=1145.576,141.150,-57.539,-178.778,6.892,148.919
C06280=1145.581,140.901,-57.519,-178.781,6.890,148.920
C06281=1145.585,140.652,-57.498,-178.784,6.889,148.920
C06282=1145.590,140.402,-57.478,-178.787,6.886,148.920
C06283=1145.595,140.153,-57.457,-178.790,6.885,148.921
C06284=1145.600,139.904,-57.436,-178.792,6.883,148.921
C06285=1145.604,139.655,-57.416,-178.795,6.881,148.921
C06286=1145.609,139.406,-57.395,-178.798,6.879,148.922
C06287=1145.614,139.156,-57.375,-178.800,6.878,148.922
C06288=1145.619,138.907,-57.355,-178.803,6.876,148.923
C06289=1145.623,138.659,-57.334,-178.806,6.873,148.923
C06290=1145.628,138.409,-57.313,-178.809,6.872,148.923
C06291=1145.633,138.160,-57.293,-178.812,6.870,148.924
C06292=1145.638,137.912,-57.273,-178.815,6.868,148.924
C06293=1145.642,137.663,-57.253,-178.817,6.867,148.925
C06294=1145.648,137.413,-57.232,-178.820,6.865,148.925
C06295=1145.652,137.164,-57.212,-178.823,6.863,148.925
C06296=1145.657,136.915,-57.192,-178.825,6.862,148.926
C06297=1145.661,136.666,-57.172,-178.829,6.859,148.926
C06298=1145.666,136.417,-57.151,-178.831,6.857,148.927
C06299=1145.671,136.168,-57.131,-178.834,6.856,148.927
C06300=1145.675,135.919,-57.110,-178.837,6.854,148.927
C06301=1145.680,135.669,-57.091,-178.839,6.852,148.928
C06302=1145.685,135.420,-57.070,-178.842,6.850,148.928
C06303=1145.690,135.172,-57.050,-178.845,6.848,148.928
C06304=1145.695,134.922,-57.030,-178.847,6.847,148.929
C06305=1145.699,134.673,-57.010,-178.851,6.844,148.929
C06306=1145.704,134.424,-56.989,-178.853,6.842,148.929
C06307=1145.709,134.174,-56.969,-178.856,6.841,148.930
C06308=1145.714,133.925,-56.949,-178.859,6.839,148.930
C06309=1145.719,133.676,-56.929,-178.861,6.837,148.931
C06310=1145.724,133.427,-56.909,-178.864,6.836,148.931
C06311=1145.728,133.179,-56.889,-178.867,6.834,148.931
C06312=1145.733,132.929,-56.869,-178.870,6.832,148.932
C06313=1145.738,132.680,-56.848,-178.872,6.831,148.932
C06314=1145.743,132.430,-56.828,-178.875,6.829,148.933
C06315=1145.747,132.181,-56.808,-178.878,6.826,148.933
C06316=1145.752,131.913,-56.787,-178.881,6.825,148.933
C06317=1145.758,131.644,-56.765,-178.884,6.823,148.934
C06318=1145.762,131.376,-56.743,-178.888,6.821,148.934
C06319=1145.768,131.107,-56.722,-178.890,6.819,148.935
C06320=1145.773,130.858,-56.702,-178.893,6.817,148.935
C06321=1145.778,130.609,-56.682,-178.896,6.816,148.936
C06322=1145.782,130.359,-56.662,-178.898,6.814,148.936
C06323=1145.787,130.110,-56.642,-178.901,6.812,148.936
C06324=1145.792,129.861,-56.623,-178.904,6.811,148.937
C06325=1145.797,129.612,-56.602,-178.907,6.809,148.937
C06326=1145.801,129.363,-56.583,-178.909,6.807,148.938
C06327=1145.806,129.114,-56.562,-178.913,6.805,148.938
C06328=1145.811,128.865,-56.543,-178.915,6.803,148.938
C06329=1145.816,128.615,-56.523,-178.918,6.801,148.939
C06330=1145.820,128.367,-56.503,-178.921,6.799,148.939
C06331=1145.825,128.117,-56.483,-178.923,6.798,148.940
C06332=1145.830,127.868,-56.464,-178.926,6.796,148.940
C06333=1145.835,127.619,-56.444,-178.929,6.794,148.940
C06334=1145.840,127.370,-56.424,-178.932,6.793,148.941
C06335=1145.844,127.120,-56.404,-178.934,6.791,148.941
C06336=1145.849,126.872,-56.384,-178.937,6.789,148.942
C06337=1145.854,126.622,-56.365,-178.940,6.788,148.942
C06338=1145.859,126.373,-56.345,-178.942,6.786,148.942
C06339=1145.864,126.123,-56.325,-178.945,6.784,148.943
C06340=1145.869,125.875,-56.305,-178.948,6.782,148.943
C06341=1145.873,125.625,-56.286,-178.951,6.781,148.943
C06342=1145.878,125.376,-56.266,-178.954,6.779,148.944
C06343=1145.883,125.127,-56.247,-178.957,6.778,148.945
C06344=1145.887,124.878,-56.227,-178.959,6.776,148.945
C06345=1145.892,124.629,-56.207,-178.962,6.774,148.945
C06346=1145.897,124.380,-56.188,-178.965,6.773,148.946
C06347=1145.902,124.130,-56.168,-178.967,6.771,148.946
C06348=1145.907,123.881,-56.149,-178.971,6.768,148.946
C06349=1145.912,123.632,-56.129,-178.973,6.767,148.947
C06350=1145.917,123.383,-56.109,-178.976,6.765,148.947
C06351=1145.921,123.134,-56.090,-178.979,6.763,148.948
C06352=1145.926,122.885,-56.071,-178.982,6.762,148.948
C06353=1145.931,122.635,-56.051,-178.984,6.760,148.948
C06354=1145.935,122.385,-56.031,-178.987,6.758,148.949
C06355=1145.941,122.137,-56.012,-178.990,6.757,148.949
C06356=1145.945,121.887,-55.993,-178.993,6.755,148.950
C06357=1145.950,121.639,-55.974,-178.995,6.753,148.950
C06358=1145.955,121.389,-55.954,-178.998,6.751,148.951
C06359=1145.960,121.139,-55.935,-179.001,6.750,148.951
C06360=1145.965,120.891,-55.915,-179.004,6.748,148.952
C06361=1145.969,120.642,-55.895,-179.007,6.747,148.952
C06362=1145.974,120.393,-55.876,-179.009,6.745,148.952
C06363=1145.979,120.143,-55.857,-179.012,6.743,148.953
C06364=1145.983,119.894,-55.837,-179.015,6.742,148.953
C06365=1145.988,119.645,-55.819,-179.018,6.740,148.954
C06366=1145.993,119.395,-55.799,-179.020,6.738,148.954
C06367=1145.998,119.146,-55.780,-179.023,6.737,148.954
C06368=1146.003,118.897,-55.760,-179.026,6.735,148.955
C06369=1146.008,118.648,-55.742,-179.028,6.733,148.955
C06370=1146.013,118.399,-55.722,-179.031,6.731,148.956
C06371=1146.017,118.149,-55.702,-179.034,6.730,148.956
C06372=1146.022,117.900,-55.684,-179.037,6.728,148.956
C06373=1146.027,117.651,-55.664,-179.040,6.727,148.957
C06374=1146.032,117.402,-55.645,-179.043,6.725,148.957
C06375=1146.036,117.153,-55.626,-179.045,6.723,148.958
C06376=1146.042,116.903,-55.607,-179.048,6.722,148.958
C06377=1146.046,116.654,-55.587,-179.051,6.720,148.959
C06378=1146.051,116.405,-55.569,-179.053,6.718,148.959
C06379=1146.056,116.156,-55.549,-179.056,6.717,148.959
C06380=1146.061,115.907,-55.530,-179.058,6.716,148.960
C06381=1146.065,115.657,-55.511,-179.061,6.714,148.960
C06382=1146.071,115.408,-55.492,-179.064,6.712,148.961
C06383=1146.075,115.159,-55.473,-179.067,6.711,148.961
C06384=1146.080,114.910,-55.454,-179.070,6.709,148.962
C06385=1146.085,114.660,-55.434,-179.072,6.708,148.962
C06386=1146.090,114.411,-55.416,-179.075,6.706,148.962
C06387=1146.095,114.162,-55.396,-179.078,6.704,148.963
C06388=1146.099,113.913,-55.378,-179.081,6.702,148.963
C06389=1146.104,113.663,-55.358,-179.083,6.701,148.964
C06390=1146.109,113.414,-55.340,-179.086,6.699,148.964
C06391=1146.114,113.165,-55.321,-179.089,6.697,148.965
C06392=1146.119,112.916,-55.301,-179.092,6.696,148.965
C06393=1146.124,112.667,-55.283,-179.095,6.694,148.966
C06394=1146.129,112.417,-55.264,-179.097,6.693,148.966
C06395=1146.133,112.168,-55.245,-179.100,6.691,148.966
C06396=1146.138,111.918,-55.226,-179.103,6.689,148.967
C06397=1146.143,111.670,-55.207,-179.106,6.688,148.967
C06398=1146.148,111.420,-55.189,-179.108,6.686,148.968
C06399=1146.152,111.171,-55.170,-179.110,6.685,148.968
C06400=1146.158,110.922,-55.150,-179.114,6.684,148.969
C06401=1146.162,110.672,-55.132,-179.116,6.682,148.969
C06402=1146.167,110.423,-55.113,-179.119,6.680,148.969
C06403=1146.172,110.174,-55.095,-179.122,6.679,148.970
C06404=1146.177,109.925,-55.075,-179.125,6.677,148.970
C06405=1146.182,109.675,-55.057,-179.127,6.675,148.971
C06406=1146.186,109.426,-55.038,-179.130,6.674,148.971
C06407=1146.191,109.177,-55.019,-179.133,6.672,148.971
C06408=1146.196,108.928,-55.001,-179.136,6.671,148.972
C06409=1146.201,108.679,-54.981,-179.139,6.669,148.973
C06410=1146.206,108.429,-54.963,-179.141,6.667,148.973
C06411=1146.211,108.180,-54.945,-179.144,6.665,148.973
C06412=1146.216,107.931,-54.925,-179.146,6.665,148.974
C06413=1146.220,107.681,-54.907,-179.149,6.663,148.974
C06414=1146.226,107.433,-54.888,-179.152,6.661,148.975
C06415=1146.230,107.183,-54.870,-179.155,6.660,148.975
C06416=1146.235,106.934,-54.851,-179.158,6.658,148.976
C06417=1146.240,106.685,-54.833,-179.160,6.657,148.976
C06418=1146.245,106.435,-54.814,-179.163,6.655,148.976
C06419=1146.249,106.186,-54.795,-179.166,6.653,148.977
C06420=1146.255,105.918,-54.775,-179.169,6.652,148.977
C06421=1146.260,105.649,-54.756,-179.172,6.650,148.978
C06422=1146.265,105.381,-54.735,-179.174,6.648,148.978
C06423=1146.270,105.113,-54.716,-179.177,6.647,148.979
C06424=1146.275,104.863,-54.698,-179.180,6.645,148.979
C06425=1146.280,104.615,-54.678,-179.183,6.644,148.980
C06426=1146.285,104.365,-54.660,-179.186,6.642,148.980
C06427=1146.290,104.115,-54.642,-179.189,6.640,148.981
C06428=1146.295,103.866,-54.623,-179.191,6.639,148.981
C06429=1146.299,103.617,-54.604,-179.193,6.638,148.981
C06430=1146.304,103.368,-54.586,-179.197,6.637,148.982
C06431=1146.309,103.118,-54.568,-179.199,6.635,148.982
C06432=1146.315,102.869,-54.550,-179.202,6.633,148.983
C06433=1146.319,102.620,-54.531,-179.205,6.631,148.983
C06434=1146.324,102.370,-54.513,-179.208,6.630,148.984
C06435=1146.329,102.121,-54.495,-179.211,6.628,148.984
C06436=1146.334,101.872,-54.477,-179.214,6.627,148.985
C06437=1146.338,101.623,-54.457,-179.216,6.626,148.985
C06438=1146.343,101.373,-54.439,-179.218,6.624,148.986
C06439=1146.348,101.124,-54.421,-179.221,6.623,148.986
C06440=1146.353,100.875,-54.403,-179.224,6.621,148.986
C06441=1146.358,100.626,-54.385,-179.227,6.620,148.987
C06442=1146.363,100.376,-54.366,-179.230,6.618,148.987
C06443=1146.368,100.126,-54.348,-179.233,6.616,148.988
C06444=1146.373,99.878,-54.330,-179.235,6.615,148.988
C06445=1146.377,99.629,-54.312,-179.237,6.614,148.989
C06446=1146.382,99.380,-54.294,-179.241,6.612,148.989
C06447=1146.387,99.130,-54.275,-179.243,6.611,148.990
C06448=1146.392,98.881,-54.257,-179.246,6.609,148.990
C06449=1146.397,98.631,-54.239,-179.249,6.607,148.991
C06450=1146.402,98.382,-54.221,-179.251,6.606,148.991
C06451=1146.407,98.133,-54.203,-179.254,6.605,148.991
C06452=1146.412,97.883,-54.185,-179.257,6.603,148.992
C06453=1146.416,97.634,-54.166,-179.260,6.602,148.993
C06454=1146.421,97.384,-54.148,-179.262,6.600,148.993
C06455=1146.426,97.135,-54.130,-179.265,6.598,148.993
C06456=1146.431,96.886,-54.113,-179.267,6.597,148.994
C06457=1146.436,96.637,-54.095,-179.270,6.596,148.994
C06458=1146.441,96.388,-54.077,-179.273,6.594,148.995
C06459=1146.446,96.139,-54.059,-179.276,6.593,148.995
C06460=1146.451,95.889,-54.041,-179.279,6.591,148.996
C06461=1146.455,95.640,-54.022,-179.281,6.589,148.996
C06462=1146.460,95.390,-54.004,-179.284,6.589,148.997
C06463=1146.465,95.141,-53.986,-179.287,6.587,148.997
C06464=1146.470,94.892,-53.968,-179.290,6.586,148.998
C06465=1146.475,94.643,-53.950,-179.292,6.584,148.998
C06466=1146.480,94.393,-53.933,-179.295,6.583,148.999
C06467=1146.485,94.144,-53.915,-179.298,6.582,148.999
C06468=1146.490,93.895,-53.897,-179.300,6.580,148.999
C06469=1146.495,93.645,-53.879,-179.303,6.578,149.000
C06470=1146.499,93.396,-53.861,-179.306,6.577,149.000
C06471=1146.504,93.147,-53.843,-179.309,6.575,149.001
C06472=1146.509,92.897,-53.825,-179.311,6.574,149.001
C06473=1146.514,92.647,-53.808,-179.314,6.573,149.002
C06474=1146.519,92.398,-53.790,-179.317,6.571,149.002
C06475=1146.524,92.149,-53.772,-179.320,6.570,149.003
C06476=1146.529,91.900,-53.754,-179.323,6.568,149.003
C06477=1146.534,91.650,-53.736,-179.325,6.567,149.004
C06478=1146.539,91.401,-53.718,-179.327,6.566,149.004
C06479=1146.544,91.152,-53.700,-179.330,6.564,149.005
C06480=1146.548,90.903,-53.683,-179.333,6.563,149.005
C06481=1146.553,90.653,-53.666,-179.336,6.562,149.006
C06482=1146.558,90.404,-53.648,-179.338,6.560,149.006
C06483=1146.563,90.155,-53.630,-179.341,6.558,149.006
C06484=1146.568,89.906,-53.612,-179.344,6.557,149.007
C06485=1146.573,89.656,-53.595,-179.347,6.555,149.007
C06486=1146.578,89.407,-53.577,-179.349,6.554,149.008
C06487=1146.583,89.157,-53.559,-179.352,6.553,149.008
C06488=1146.587,88.908,-53.542,-179.355,6.551,149.009
C06489=1146.592,88.659,-53.524,-179.358,6.550,149.009
C06490=1146.597,88.410,-53.506,-179.360,6.549,149.010
C06491=1146.602,88.160,-53.489,-179.363,6.547,149.010
C06492=1146.607,87.911,-53.471,-179.366,6.546,149.011
C06493=1146.612,87.661,-53.454,-179.369,6.544,149.011
C06494=1146.617,87.412,-53.436,-179.371,6.543,149.012
C06495=1146.622,87.163,-53.418,-179.374,6.542,149.012
C06496=1146.627,86.913,-53.401,-179.377,6.540,149.013
C06497=1146.632,86.664,-53.383,-179.379,6.539,149.013
C06498=1146.636,86.414,-53.366,-179.382,6.538,149.014
C06499=1146.642,86.166,-53.349,-179.384,6.536,149.014
C06500=1146.647,85.916,-53.331,-179.388,6.535,149.015
C06501=1146.652,85.667,-53.313,-179.390,6.533,149.015
C06502=1146.656,85.417,-53.297,-179.392,6.532,149.016
C06503=1146.661,85.168,-53.279,-179.395,6.531,149.016
C06504=1146.666,84.918,-53.261,-179.398,6.529,149.017
C06505=1146.671,84.670,-53.244,-179.401,6.528,149.017
C06506=1146.676,84.420,-53.227,-179.403,6.527,149.018
C06507=1146.681,84.171,-53.209,-179.406,6.525,149.018
C06508=1146.685,83.921,-53.192,-179.409,6.524,149.019
C06509=1146.690,83.672,-53.174,-179.412,6.522,149.019
C06510=1146.696,83.423,-53.157,-179.414,6.521,149.019
C06511=1146.701,83.173,-53.140,-179.417,6.520,149.020
C06512=1146.705,82.924,-53.123,-179.420,6.518,149.021
C06513=1146.711,82.674,-53.105,-179.422,6.517,149.021
C06514=1146.715,82.426,-53.088,-179.425,6.516,149.021
C06515=1146.720,82.176,-53.071,-179.428,6.514,149.022
C06516=1146.725,81.926,-53.053,-179.431,6.513,149.022
C06517=1146.729,81.677,-53.036,-179.433,6.512,149.023
C06518=1146.735,81.428,-53.019,-179.436,6.510,149.023
C06519=1146.740,81.178,-53.002,-179.439,6.509,149.024
C06520=1146.745,80.929,-52.984,-179.441,6.508,149.024
C06521=1146.750,80.680,-52.967,-179.444,6.506,149.025
C06522=1146.754,80.430,-52.951,-179.447,6.505,149.025
C06523=1146.759,80.181,-52.933,-179.450,6.504,149.026
C06524=1146.765,79.913,-52.914,-179.452,6.503,149.026
C06525=1146.770,79.644,-52.896,-179.455,6.501,149.027
C06526=1146.776,79.376,-52.878,-179.458,6.500,149.027
C06527=1146.781,79.107,-52.859,-179.461,6.498,149.028
C06528=1146.786,78.858,-52.842,-179.464,6.497,149.028
C06529=1146.791,78.608,-52.824,-179.467,6.495,149.029
C06530=1146.796,78.360,-52.808,-179.469,6.494,149.029
C06531=1146.801,78.110,-52.791,-179.472,6.493,149.030
C06532=1146.805,77.860,-52.774,-179.475,6.491,149.030
C06533=1146.811,77.611,-52.757,-179.477,6.490,149.031
C06534=1146.815,77.362,-52.740,-179.480,6.489,149.031
C06535=1146.821,77.113,-52.723,-179.483,6.487,149.032
C06536=1146.825,76.863,-52.706,-179.485,6.487,149.032
C06537=1146.830,76.613,-52.689,-179.488,6.485,149.033
C06538=1146.835,76.364,-52.672,-179.491,6.484,149.033
C06539=1146.841,76.115,-52.655,-179.493,6.483,149.034
C06540=1146.845,75.865,-52.638,-179.496,6.481,149.034
C06541=1146.850,75.616,-52.621,-179.499,6.479,149.035
C06542=1146.854,75.367,-52.604,-179.501,6.479,149.035
C06543=1146.860,75.118,-52.588,-179.504,6.477,149.036
C06544=1146.865,74.868,-52.570,-179.507,6.476,149.036
C06545=1146.869,74.619,-52.554,-179.509,6.475,149.037
C06546=1146.875,74.369,-52.537,-179.512,6.473,149.037
C06547=1146.880,74.120,-52.520,-179.515,6.472,149.038
C06548=1146.885,73.870,-52.503,-179.518,6.471,149.038
C06549=1146.889,73.621,-52.486,-179.520,6.470,149.039
C06550=1146.894,73.372,-52.470,-179.523,6.468,149.039
C06551=1146.900,73.122,-52.453,-179.525,6.467,149.040
C06552=1146.904,72.873,-52.436,-179.528,6.466,149.040
C06553=1146.909,72.624,-52.420,-179.531,6.464,149.041
C06554=1146.914,72.374,-52.402,-179.533,6.463,149.041
C06555=1146.919,72.125,-52.386,-179.537,6.462,149.042
C06556=1146.925,71.875,-52.369,-179.539,6.460,149.042
C06557=1146.929,71.626,-52.352,-179.541,6.459,149.043
C06558=1146.934,71.377,-52.335,-179.545,6.458,149.043
C06559=1146.939,71.127,-52.318,-179.547,6.457,149.044
C06560=1146.944,70.878,-52.302,-179.550,6.456,149.044
C06561=1146.948,70.628,-52.285,-179.553,6.454,149.045
C06562=1146.954,70.379,-52.269,-179.555,6.453,149.045
C06563=1146.959,70.129,-52.252,-179.558,6.452,149.046
C06564=1146.963,69.880,-52.236,-179.561,6.450,149.046
C06565=1146.969,69.631,-52.219,-179.563,6.450,149.047
C06566=1146.974,69.381,-52.202,-179.566,6.448,149.047
C06567=1146.979,69.132,-52.186,-179.569,6.446,149.048
C06568=1146.983,68.883,-52.169,-179.571,6.446,149.048
C06569=1146.988,68.633,-52.153,-179.574,6.444,149.049
C06570=1146.994,68.384,-52.136,-179.576,6.443,149.049
C06571=1146.998,68.134,-52.120,-179.579,6.442,149.050
C06572=1147.003,67.885,-52.103,-179.582,6.440,149.050
C06573=1147.008,67.636,-52.087,-179.584,6.439,149.051
C06574=1147.013,67.386,-52.070,-179.587,6.438,149.051
C06575=1147.019,67.137,-52.054,-179.590,6.437,149.052
C06576=1147.023,66.887,-52.037,-179.592,6.436,149.052
C06577=1147.028,66.639,-52.021,-179.596,6.434,149.053
C06578=1147.033,66.388,-52.005,-179.598,6.434,149.053
C06579=1147.038,66.139,-51.988,-179.600,6.432,149.054
C06580=1147.043,65.890,-51.971,-179.603,6.431,149.055
C06581=1147.048,65.640,-51.955,-179.606,6.430,149.055
C06582=1147.053,65.391,-51.939,-179.609,6.428,149.055
C06583=1147.058,65.141,-51.922,-179.611,6.428,149.056
C06584=1147.063,64.893,-51.906,-179.614,6.426,149.056
C06585=1147.068,64.642,-51.889,-179.616,6.425,149.057
C06586=1147.073,64.393,-51.873,-179.619,6.424,149.058
C06587=1147.078,64.144,-51.857,-179.622,6.422,149.058
C06588=1147.082,63.894,-51.841,-179.624,6.421,149.058
C06589=1147.088,63.645,-51.824,-179.627,6.420,149.059
C06590=1147.092,63.395,-51.808,-179.630,6.419,149.060
C06591=1147.097,63.146,-51.792,-179.632,6.417,149.060
C06592=1147.102,62.897,-51.775,-179.636,6.416,149.061
C06593=1147.108,62.647,-51.759,-179.638,6.415,149.061
C06594=1147.113,62.398,-51.742,-179.640,6.414,149.062
C06595=1147.118,62.148,-51.727,-179.643,6.413,149.062
C06596=1147.122,61.899,-51.710,-179.646,6.412,149.063
C06597=1147.127,61.650,-51.694,-179.648,6.411,149.063
C06598=1147.132,61.400,-51.678,-179.651,6.409,149.064
C06599=1147.137,61.151,-51.662,-179.654,6.408,149.064
C06600=1147.143,60.902,-51.646,-179.657,6.407,149.065
C06601=1147.147,60.652,-51.629,-179.659,6.406,149.065
C06602=1147.153,60.403,-51.614,-179.662,6.405,149.066
C06603=1147.157,60.153,-51.597,-179.665,6.403,149.066
C06604=1147.162,59.904,-51.582,-179.667,6.403,149.067
C06605=1147.167,59.654,-51.565,-179.670,6.401,149.067
C06606=1147.172,59.405,-51.549,-179.672,6.400,149.068
C06607=1147.177,59.155,-51.533,-179.675,6.399,149.068
C06608=1147.182,58.906,-51.517,-179.678,6.397,149.069
C06609=1147.187,58.656,-51.501,-179.680,6.397,149.069
C06610=1147.192,58.407,-51.485,-179.683,6.395,149.070
C06611=1147.197,58.158,-51.469,-179.685,6.394,149.070
C06612=1147.202,57.908,-51.453,-179.689,6.393,149.071
C06613=1147.207,57.659,-51.437,-179.691,6.392,149.071
C06614=1147.212,57.409,-51.421,-179.693,6.390,149.072
C06615=1147.217,57.160,-51.405,-179.696,6.390,149.073
C06616=1147.223,56.911,-51.389,-179.699,6.388,149.073
C06617=1147.227,56.660,-51.373,-179.702,6.388,149.074
C06618=1147.232,56.412,-51.357,-179.704,6.386,149.074
C06619=1147.237,56.162,-51.341,-179.706,6.385,149.075
C06620=1147.243,55.912,-51.325,-179.710,6.384,149.075
C06621=1147.247,55.664,-51.310,-179.712,6.382,149.076
C06622=1147.252,55.414,-51.294,-179.715,6.381,149.076
C06623=1147.257,55.164,-51.278,-179.718,6.380,149.077
C06624=1147.262,54.915,-51.262,-179.720,6.379,149.077
C06625=1147.267,54.665,-51.246,-179.723,6.378,149.078
C06626=1147.272,54.416,-51.230,-179.725,6.377,149.078
C06627=1147.278,54.167,-51.215,-179.728,6.376,149.079
C06628=1147.283,53.897,-51.197,-179.731,6.375,149.079
C06629=1147.288,53.629,-51.180,-179.733,6.373,149.080
C06630=1147.294,53.360,-51.163,-179.737,6.372,149.080
C06631=1147.299,53.092,-51.147,-179.739,6.371,149.081
C06632=1147.303,52.842,-51.131,-179.742,6.370,149.082
C06633=1147.309,52.593,-51.115,-179.745,6.368,149.082
C06634=1147.314,52.344,-51.099,-179.747,6.368,149.083
C06635=1147.319,52.095,-51.083,-179.750,6.366,149.083
C06636=1147.324,51.844,-51.067,-179.752,6.365,149.084
C06637=1147.329,51.595,-51.052,-179.756,6.364,149.084
C06638=1147.334,51.346,-51.037,-179.758,6.363,149.085
C06639=1147.339,51.096,-51.020,-179.761,6.362,149.085
C06640=1147.344,50.847,-51.005,-179.763,6.361,149.086
C06641=1147.349,50.598,-50.990,-179.766,6.360,149.086
C06642=1147.353,50.348,-50.974,-179.769,6.359,149.087
C06643=1147.359,50.098,-50.958,-179.771,6.358,149.087
C06644=1147.364,49.849,-50.942,-179.773,6.357,149.088
C06645=1147.369,49.600,-50.927,-179.776,6.356,149.088
C06646=1147.374,49.350,-50.911,-179.779,6.354,149.089
C06647=1147.379,49.100,-50.896,-179.781,6.354,149.089
C06648=1147.384,48.851,-50.880,-179.784,6.352,149.090
C06649=1147.389,48.602,-50.865,-179.786,6.351,149.090
C06650=1147.394,48.352,-50.849,-179.790,6.350,149.091
C06651=1147.399,48.102,-50.834,-179.792,6.349,149.092
C06652=1147.404,47.853,-50.819,-179.795,6.348,149.092
C06653=1147.409,47.604,-50.803,-179.797,6.347,149.093
C06654=1147.414,47.354,-50.787,-179.800,6.346,149.093
C06655=1147.419,47.105,-50.772,-179.803,6.345,149.094
C06656=1147.424,46.855,-50.757,-179.805,6.343,149.094
C06657=1147.429,46.606,-50.741,-179.808,6.343,149.095
C06658=1147.434,46.356,-50.726,-179.811,6.341,149.095
C06659=1147.439,46.107,-50.710,-179.813,6.341,149.096
C06660=1147.444,45.857,-50.695,-179.816,6.339,149.096
C06661=1147.449,45.608,-50.680,-179.818,6.338,149.097
C06662=1147.454,45.359,-50.664,-179.820,6.338,149.097
C06663=1147.459,45.109,-50.648,-179.824,6.336,149.098
C06664=1147.464,44.860,-50.633,-179.826,6.335,149.098
C06665=1147.469,44.610,-50.617,-179.829,6.334,149.099
C06666=1147.474,44.361,-50.602,-179.831,6.333,149.100
C06667=1147.479,44.112,-50.587,-179.834,6.332,149.100
C06668=1147.485,43.862,-50.572,-179.837,6.331,149.101
C06669=1147.489,43.612,-50.557,-179.839,6.330,149.101
C06670=1147.494,43.363,-50.541,-179.842,6.329,149.102
C06671=1147.499,43.113,-50.526,-179.844,6.328,149.102
C06672=1147.504,42.864,-50.510,-179.847,6.327,149.103
C06673=1147.509,42.615,-50.495,-179.850,6.326,149.103
C06674=1147.515,42.365,-50.481,-179.852,6.325,149.104
C06675=1147.519,42.115,-50.465,-179.855,6.324,149.104
C06676=1147.524,41.866,-50.450,-179.858,6.322,149.105
C06677=1147.530,41.616,-50.434,-179.860,6.322,149.105
C06678=1147.534,41.367,-50.420,-179.863,6.320,149.106
C06679=1147.540,41.117,-50.404,-179.865,6.319,149.107
C06680=1147.544,40.868,-50.389,-179.868,6.319,149.107
C06681=1147.550,40.619,-50.374,-179.871,6.317,149.108
C06682=1147.555,40.369,-50.359,-179.873,6.317,149.108
C06683=1147.560,40.120,-50.344,-179.876,6.315,149.109
C06684=1147.564,39.870,-50.328,-179.878,6.314,149.109
C06685=1147.570,39.620,-50.313,-179.880,6.314,149.110
C06686=1147.575,39.371,-50.299,-179.884,6.312,149.110
C06687=1147.580,39.121,-50.283,-179.886,6.311,149.111
C06688=1147.585,38.872,-50.268,-179.889,6.310,149.111
C06689=1147.590,38.622,-50.253,-179.891,6.309,149.112
C06690=1147.595,38.373,-50.238,-179.894,6.308,149.112
C06691=1147.600,38.124,-50.223,-179.897,6.307,149.113
C06692=1147.605,37.874,-50.208,-179.899,6.306,149.114
C06693=1147.610,37.625,-50.193,-179.902,6.305,149.114
C06694=1147.616,37.375,-50.178,-179.904,6.304,149.115
C06695=1147.620,37.126,-50.163,-179.907,6.303,149.115
C06696=1147.626,36.876,-50.148,-179.910,6.302,149.116
C06697=1147.631,36.627,-50.133,-179.912,6.301,149.116
C06698=1147.635,36.378,-50.118,-179.915,6.300,149.117
C06699=1147.641,36.128,-50.104,-179.917,6.299,149.117
C06700=1147.645,35.878,-50.088,-179.920,6.298,149.118
C06701=1147.651,35.628,-50.073,-179.923,6.297,149.118
C06702=1147.655,35.379,-50.058,-179.925,6.296,149.119
C06703=1147.660,35.130,-50.043,-179.928,6.295,149.120
C06704=1147.666,34.880,-50.029,-179.930,6.294,149.120
C06705=1147.670,34.630,-50.014,-179.933,6.294,149.121
C06706=1147.675,34.381,-49.999,-179.936,6.292,149.121
C06707=1147.681,34.131,-49.984,-179.938,6.291,149.122
C06708=1147.686,33.882,-49.969,-179.941,6.290,149.122
C06709=1147.690,33.633,-49.954,-179.943,6.289,149.123
C06710=1147.696,33.383,-49.940,-179.946,6.289,149.123
C06711=1147.701,33.133,-49.925,-179.949,6.287,149.124
C06712=1147.706,32.884,-49.910,-179.951,6.287,149.125
C06713=1147.712,32.634,-49.896,-179.953,6.286,149.125
C06714=1147.717,32.385,-49.881,-179.956,6.284,149.125
C06715=1147.722,32.136,-49.866,-179.959,6.284,149.126
C06716=1147.726,31.887,-49.851,-179.962,6.282,149.127
C06717=1147.732,31.636,-49.837,-179.964,6.282,149.127
C06718=1147.737,31.387,-49.822,-179.966,6.281,149.128
C06719=1147.741,31.138,-49.807,-179.969,6.279,149.128
C06720=1147.746,30.888,-49.793,-179.972,6.279,149.129
C06721=1147.752,30.639,-49.777,-179.974,6.278,149.129
C06722=1147.757,30.389,-49.763,-179.977,6.277,149.130
C06723=1147.762,30.139,-49.749,-179.979,6.276,149.130
C06724=1147.766,29.890,-49.734,-179.982,6.275,149.131
C06725=1147.772,29.640,-49.719,-179.985,6.274,149.132
C06726=1147.777,29.390,-49.705,-179.987,6.273,149.132
C06727=1147.782,29.141,-49.690,-179.990,6.272,149.133
C06728=1147.787,28.892,-49.676,-179.992,6.271,149.133
C06729=1147.792,28.642,-49.661,-179.995,6.270,149.134
C06730=1147.798,28.392,-49.647,-179.998,6.269,149.134
C06731=1147.803,28.143,-49.632,180.000,6.268,149.135
C06732=1147.808,27.874,-49.617,179.997,6.267,149.135
C06733=1147.813,27.605,-49.601,179.994,6.266,149.136
C06734=1147.819,27.336,-49.585,179.992,6.265,149.137
C06735=1147.824,27.067,-49.569,179.989,6.264,149.137
C06736=1147.829,26.818,-49.555,179.987,6.263,149.138
C06737=1147.834,26.568,-49.540,179.983,6.262,149.138
C06738=1147.840,26.319,-49.527,179.981,6.261,149.139
C06739=1147.844,26.070,-49.512,179.979,6.261,149.139
C06740=1147.850,25.820,-49.497,179.976,6.259,149.140
C06741=1147.855,25.570,-49.482,179.973,6.259,149.141
C06742=1147.860,25.320,-49.468,179.971,6.258,149.141
C06743=1147.865,25.071,-49.454,179.968,6.256,149.141
C06744=1147.870,24.821,-49.440,179.966,6.256,149.142
C06745=1147.875,24.573,-49.425,179.963,6.255,149.143
C06746=1147.880,24.323,-49.411,179.961,6.254,149.143
C06747=1147.885,24.073,-49.396,179.958,6.253,149.144
C06748=1147.890,23.823,-49.382,179.955,6.252,149.144
C06749=1147.895,23.574,-49.368,179.953,6.252,149.145
C06750=1147.900,23.324,-49.354,179.950,6.250,149.145
C06751=1147.905,23.075,-49.340,179.948,6.249,149.146
C06752=1147.910,22.825,-49.325,179.946,6.249,149.146
C06753=1147.916,22.575,-49.311,179.942,6.247,149.147
C06754=1147.921,22.326,-49.296,179.940,6.247,149.148
C06755=1147.926,22.076,-49.282,179.938,6.246,149.148
C06756=1147.931,21.827,-49.267,179.935,6.244,149.149
C06757=1147.936,21.578,-49.253,179.933,6.244,149.149
C06758=1147.941,21.328,-49.239,179.930,6.243,149.150
C06759=1147.946,21.078,-49.224,179.928,6.242,149.150
C06760=1147.952,20.829,-49.211,179.925,6.241,149.151
C06761=1147.956,20.580,-49.196,179.922,6.240,149.151
C06762=1147.961,20.330,-49.182,179.920,6.240,149.152
C06763=1147.966,20.080,-49.168,179.917,6.238,149.153
C06764=1147.971,19.830,-49.153,179.914,6.238,149.153
C06765=1147.977,19.581,-49.140,179.912,6.237,149.154
C06766=1147.981,19.331,-49.127,179.910,6.236,149.154
C06767=1147.986,19.082,-49.112,179.907,6.235,149.155
C06768=1147.991,18.832,-49.098,179.905,6.234,149.155
C06769=1147.997,18.583,-49.084,179.902,6.234,149.156
C06770=1148.002,18.333,-49.070,179.899,6.232,149.157
C06771=1148.007,18.084,-49.056,179.897,6.231,149.157
C06772=1148.012,17.835,-49.042,179.894,6.231,149.158
C06773=1148.017,17.585,-49.027,179.892,6.230,149.158
C06774=1148.022,17.335,-49.013,179.889,6.229,149.159
C06775=1148.027,17.085,-48.999,179.887,6.228,149.159
C06776=1148.033,16.836,-48.985,179.884,6.227,149.160
C06777=1148.038,16.586,-48.971,179.882,6.226,149.160
C06778=1148.042,16.337,-48.958,179.879,6.225,149.161
C06779=1148.048,16.088,-48.944,179.877,6.224,149.162
C06780=1148.053,15.838,-48.929,179.874,6.224,149.162
C06781=1148.058,15.588,-48.915,179.872,6.223,149.163
C06782=1148.063,15.339,-48.901,179.869,6.222,149.163
C06783=1148.069,15.089,-48.888,179.866,6.221,149.164
C06784=1148.073,14.839,-48.873,179.864,6.220,149.164
C06785=1148.078,14.591,-48.860,179.861,6.220,149.165
C06786=1148.083,14.341,-48.846,179.859,6.218,149.165
C06787=1148.089,14.090,-48.832,179.856,6.218,149.166
C06788=1148.094,13.841,-48.818,179.854,6.217,149.167
C06789=1148.099,13.592,-48.804,179.851,6.216,149.167
C06790=1148.104,13.342,-48.790,179.848,6.215,149.168
C06791=1148.109,13.093,-48.777,179.846,6.214,149.168
C06792=1148.114,12.843,-48.763,179.844,6.214,149.169
C06793=1148.119,12.593,-48.749,179.841,6.213,149.169
C06794=1148.125,12.344,-48.735,179.838,6.212,149.170
C06795=1148.130,12.094,-48.721,179.836,6.211,149.170
C06796=1148.134,11.845,-48.708,179.833,6.210,149.171
C06797=1148.140,11.596,-48.694,179.831,6.209,149.172
C06798=1148.145,11.345,-48.680,179.828,6.208,149.172
C06799=1148.150,11.096,-48.666,179.826,6.207,149.173
C06800=1148.155,10.847,-48.652,179.824,6.207,149.173
C06801=1148.160,10.596,-48.639,179.821,6.206,149.174
C06802=1148.165,10.347,-48.625,179.819,6.205,149.174
C06803=1148.170,10.098,-48.611,179.816,6.204,149.175
C06804=1148.176,9.848,-48.598,179.813,6.203,149.175
C06805=1148.180,9.599,-48.584,179.811,6.203,149.176
C06806=1148.186,9.348,-48.570,179.809,6.202,149.177
C06807=1148.191,9.100,-48.557,179.805,6.201,149.177
C06808=1148.196,8.850,-48.543,179.803,6.200,149.178
C06809=1148.201,8.600,-48.529,179.801,6.199,149.178
C06810=1148.206,8.351,-48.516,179.798,6.199,149.179
C06811=1148.211,8.101,-48.503,179.796,6.198,149.179
C06812=1148.216,7.852,-48.488,179.793,6.197,149.180
C06813=1148.221,7.602,-48.475,179.791,6.196,149.181
C06814=1148.226,7.353,-48.461,179.788,6.195,149.181
C06815=1148.232,7.102,-48.448,179.786,6.195,149.182
C06816=1148.237,6.854,-48.435,179.783,6.194,149.182
C06817=1148.242,6.603,-48.421,179.780,6.192,149.183
C06818=1148.247,6.354,-48.407,179.778,6.192,149.184
C06819=1148.252,6.104,-48.394,179.776,6.191,149.184
C06820=1148.257,5.855,-48.380,179.773,6.190,149.184
C06821=1148.263,5.605,-48.367,179.771,6.190,149.185
C06822=1148.268,5.356,-48.353,179.768,6.188,149.186
C06823=1148.273,5.106,-48.340,179.765,6.188,149.186
C06824=1148.278,4.857,-48.326,179.763,6.187,149.187
C06825=1148.283,4.607,-48.313,179.761,6.187,149.187
C06826=1148.288,4.358,-48.299,179.758,6.186,149.188
C06827=1148.293,4.108,-48.286,179.755,6.185,149.189
C06828=1148.299,3.858,-48.273,179.753,6.184,149.189
C06829=1148.303,3.609,-48.259,179.751,6.183,149.190
C06830=1148.309,3.359,-48.246,179.748,6.183,149.190
C06831=1148.313,3.110,-48.232,179.746,6.182,149.191
C06832=1148.319,2.860,-48.219,179.743,6.181,149.191
C06833=1148.323,2.610,-48.206,179.741,6.180,149.192
C06834=1148.329,2.361,-48.192,179.738,6.179,149.192
C06835=1148.334,2.111,-48.179,179.736,6.178,149.193
C06836=1148.340,1.842,-48.165,179.733,6.178,149.194
C06837=1148.345,1.572,-48.150,179.730,6.176,149.194
C06838=1148.351,1.303,-48.135,179.728,6.176,149.195
C06839=1148.356,1.033,-48.122,179.725,6.175,149.195
C06840=1148.362,0.784,-48.108,179.723,6.175,149.196
C06841=1148.366,0.535,-48.095,179.720,6.173,149.197
C06842=1148.372,0.285,-48.082,179.717,6.173,149.197
C06843=1148.377,0.035,-48.069,179.715,6.172,149.198
C06844=1148.382,-0.215,-48.055,179.713,6.171,149.198
C06845=1148.387,-0.464,-48.042,179.710,6.171,149.199
C06846=1148.392,-0.714,-48.029,179.708,6.170,149.199
C06847=1148.397,-0.963,-48.016,179.705,6.168,149.200
C06848=1148.403,-1.212,-48.002,179.702,6.168,149.201
C06849=1148.407,-1.463,-47.989,179.700,6.167,149.201
C06850=1148.413,-1.712,-47.976,179.697,6.167,149.202
C06851=1148.418,-1.962,-47.963,179.695,6.166,149.202
C06852=1148.423,-2.211,-47.950,179.693,6.166,149.203
C06853=1148.428,-2.460,-47.936,179.690,6.165,149.203
C06854=1148.433,-2.711,-47.923,179.687,6.164,149.204
C06855=1148.439,-2.960,-47.910,179.685,6.163,149.204
C06856=1148.444,-3.209,-47.898,179.683,6.162,149.205
C06857=1148.448,-3.459,-47.885,179.680,6.161,149.206
C06858=1148.454,-3.709,-47.871,179.678,6.161,149.206
C06859=1148.459,-3.958,-47.858,179.675,6.160,149.207
C06860=1148.464,-4.208,-47.845,179.673,6.159,149.207
C06861=1148.470,-4.457,-47.832,179.670,6.158,149.208
C06862=1148.474,-4.707,-47.819,179.668,6.157,149.208
C06863=1148.480,-4.957,-47.806,179.665,6.157,149.209
C06864=1148.485,-5.206,-47.793,179.663,6.156,149.210
C06865=1148.490,-5.456,-47.780,179.660,6.156,149.210
C06866=1148.495,-5.706,-47.767,179.658,6.155,149.211
C06867=1148.501,-5.955,-47.754,179.656,6.154,149.211
C06868=1148.505,-6.205,-47.741,179.653,6.154,149.212
C06869=1148.511,-6.454,-47.728,179.650,6.152,149.212
C06870=1148.516,-6.704,-47.715,179.648,6.152,149.213
C06871=1148.520,-6.954,-47.702,179.646,6.151,149.214
C06872=1148.526,-7.203,-47.689,179.643,6.150,149.214
C06873=1148.531,-7.453,-47.676,179.641,6.150,149.215
C06874=1148.536,-7.703,-47.663,179.638,6.149,149.215
C06875=1148.542,-7.952,-47.650,179.636,6.148,149.216
C06876=1148.547,-8.202,-47.637,179.633,6.148,149.217
C06877=1148.552,-8.451,-47.625,179.631,6.147,149.217
C06878=1148.556,-8.701,-47.612,179.628,6.145,149.217
C06879=1148.562,-8.951,-47.599,179.626,6.145,149.218
C06880=1148.567,-9.200,-47.586,179.623,6.144,149.219
C06881=1148.572,-9.450,-47.573,179.621,6.144,149.219
C06882=1148.577,-9.699,-47.561,179.619,6.143,149.220
C06883=1148.583,-9.949,-47.547,179.616,6.143,149.220
C06884=1148.588,-10.199,-47.535,179.614,6.142,149.221
C06885=1148.593,-10.449,-47.522,179.611,6.141,149.222
C06886=1148.598,-10.698,-47.510,179.609,6.141,149.222
C06887=1148.604,-10.948,-47.497,179.607,6.140,149.223
C06888=1148.608,-11.198,-47.484,179.604,6.139,149.223
C06889=1148.614,-11.447,-47.471,179.601,6.138,149.224
C06890=1148.619,-11.696,-47.459,179.599,6.137,149.224
C06891=1148.624,-11.946,-47.446,179.597,6.136,149.225
C06892=1148.630,-12.195,-47.433,179.594,6.136,149.226
C06893=1148.634,-12.445,-47.420,179.592,6.135,149.226
C06894=1148.640,-12.695,-47.408,179.589,6.135,149.227
C06895=1148.645,-12.945,-47.395,179.587,6.134,149.227
C06896=1148.650,-13.194,-47.383,179.584,6.134,149.228
C06897=1148.654,-13.444,-47.370,179.582,6.133,149.228
C06898=1148.660,-13.694,-47.357,179.580,6.132,149.229
C06899=1148.665,-13.943,-47.344,179.577,6.132,149.230
C06900=1148.671,-14.193,-47.332,179.575,6.131,149.230
C06901=1148.676,-14.442,-47.319,179.572,6.130,149.231
C06902=1148.680,-14.692,-47.306,179.570,6.129,149.231
C06903=1148.686,-14.942,-47.294,179.567,6.128,149.232
C06904=1148.691,-15.191,-47.282,179.565,6.127,149.232
C06905=1148.696,-15.441,-47.269,179.562,6.127,149.233
C06906=1148.702,-15.690,-47.256,179.560,6.126,149.233
C06907=1148.706,-15.940,-47.243,179.557,6.126,149.234
C06908=1148.712,-16.190,-47.231,179.555,6.125,149.235
C06909=1148.717,-16.440,-47.219,179.553,6.124,149.235
C06910=1148.722,-16.689,-47.206,179.550,6.124,149.236
C06911=1148.727,-16.938,-47.194,179.548,6.123,149.236
C06912=1148.733,-17.188,-47.182,179.545,6.123,149.237
C06913=1148.737,-17.438,-47.169,179.543,6.122,149.237
C06914=1148.742,-17.688,-47.156,179.541,6.121,149.238
C06915=1148.748,-17.938,-47.144,179.538,6.121,149.239
C06916=1148.753,-18.187,-47.132,179.536,6.120,149.239
C06917=1148.758,-18.436,-47.119,179.534,6.119,149.240
C06918=1148.763,-18.686,-47.107,179.531,6.119,149.240
C06919=1148.769,-18.935,-47.094,179.528,6.117,149.241
C06920=1148.774,-19.185,-47.082,179.526,6.117,149.241
C06921=1148.779,-19.435,-47.070,179.523,6.116,149.242
C06922=1148.784,-19.685,-47.057,179.521,6.115,149.243
C06923=1148.790,-19.935,-47.045,179.518,6.115,149.243
C06924=1148.795,-20.184,-47.032,179.516,6.114,149.244
C06925=1148.800,-20.434,-47.019,179.514,6.114,149.244
C06926=1148.805,-20.684,-47.007,179.511,6.113,149.245
C06927=1148.811,-20.933,-46.995,179.509,6.112,149.245
C06928=1148.815,-21.182,-46.984,179.507,6.112,149.246
C06929=1148.820,-21.432,-46.971,179.504,6.111,149.247
C06930=1148.826,-21.681,-46.958,179.502,6.110,149.247
C06931=1148.830,-21.932,-46.946,179.500,6.110,149.248
C06932=1148.836,-22.181,-46.934,179.497,6.109,149.248
C06933=1148.841,-22.431,-46.922,179.495,6.108,149.249
C06934=1148.846,-22.680,-46.909,179.492,6.108,149.250
C06935=1148.851,-22.930,-46.897,179.490,6.107,149.250
C06936=1148.857,-23.180,-46.885,179.488,6.106,149.251
C06937=1148.862,-23.430,-46.873,179.485,6.106,149.251
C06938=1148.867,-23.679,-46.860,179.483,6.105,149.252
C06939=1148.873,-23.929,-46.848,179.480,6.105,149.252
C06940=1148.878,-24.199,-46.835,179.478,6.104,149.253
C06941=1148.884,-24.468,-46.822,179.475,6.104,149.254
C06942=1148.890,-24.739,-46.808,179.472,6.102,149.254
C06943=1148.895,-25.009,-46.795,179.470,6.102,149.255
C06944=1148.900,-25.258,-46.783,179.467,6.101,149.255
C06945=1148.905,-25.508,-46.771,179.465,6.100,149.256
C06946=1148.911,-25.758,-46.758,179.462,6.100,149.257
C06947=1148.915,-26.007,-46.747,179.460,6.099,149.257
C06948=1148.921,-26.257,-46.735,179.457,6.099,149.258
C06949=1148.926,-26.507,-46.723,179.455,6.098,149.258
C06950=1148.931,-26.757,-46.711,179.453,6.097,149.259
C06951=1148.936,-27.006,-46.698,179.450,6.097,149.259
C06952=1148.942,-27.256,-46.686,179.448,6.096,149.260
C06953=1148.946,-27.505,-46.675,179.446,6.095,149.261
C06954=1148.952,-27.755,-46.662,179.443,6.095,149.261
C06955=1148.957,-28.005,-46.650,179.441,6.094,149.262
C06956=1148.962,-28.255,-46.638,179.439,6.093,149.262
C06957=1148.968,-28.504,-46.626,179.436,6.093,149.263
C06958=1148.972,-28.754,-46.615,179.434,6.092,149.263
C06959=1148.978,-29.003,-46.603,179.432,6.091,149.264
C06960=1148.983,-29.253,-46.590,179.429,6.091,149.265
C06961=1148.988,-29.503,-46.578,179.427,6.090,149.265
C06962=1148.994,-29.753,-46.566,179.424,6.090,149.266
C06963=1148.998,-30.002,-46.554,179.422,6.089,149.266
C06964=1149.004,-30.251,-46.543,179.419,6.089,149.267
C06965=1149.010,-30.501,-46.531,179.417,6.088,149.267
C06966=1149.015,-30.751,-46.519,179.415,6.088,149.268
C06967=1149.019,-31.000,-46.507,179.413,6.087,149.269
C06968=1149.025,-31.250,-46.495,179.411,6.087,149.269
C06969=1149.030,-31.500,-46.483,179.408,6.086,149.270
C06970=1149.036,-31.750,-46.471,179.406,6.085,149.270
C06971=1149.040,-31.999,-46.459,179.403,6.085,149.271
C06972=1149.045,-32.249,-46.447,179.401,6.084,149.271
C06973=1149.051,-32.498,-46.436,179.398,6.084,149.272
C06974=1149.056,-32.748,-46.424,179.396,6.083,149.273
C06975=1149.061,-32.998,-46.412,179.394,6.082,149.273
C06976=1149.066,-33.247,-46.400,179.391,6.082,149.274
C06977=1149.072,-33.497,-46.388,179.389,6.081,149.274
C06978=1149.077,-33.746,-46.377,179.386,6.081,149.275
C06979=1149.082,-33.996,-46.365,179.384,6.080,149.275
C06980=1149.088,-34.246,-46.353,179.381,6.079,149.276
C06981=1149.092,-34.496,-46.342,179.379,6.079,149.277
C06982=1149.098,-34.746,-46.330,179.377,6.078,149.277
C06983=1149.103,-34.995,-46.317,179.374,6.077,149.278
C06984=1149.108,-35.245,-46.306,179.372,6.077,149.278
C06985=1149.113,-35.495,-46.294,179.370,6.076,149.279
C06986=1149.119,-35.744,-46.283,179.367,6.075,149.279
C06987=1149.124,-35.993,-46.271,179.365,6.075,149.280
C06988=1149.129,-36.243,-46.260,179.363,6.074,149.281
C06989=1149.135,-36.493,-46.248,179.361,6.074,149.281
C06990=1149.139,-36.743,-46.236,179.358,6.074,149.282
C06991=1149.145,-36.993,-46.225,179.356,6.073,149.282
C06992=1149.150,-37.243,-46.213,179.353,6.073,149.283
C06993=1149.155,-37.492,-46.202,179.351,6.072,149.283
C06994=1149.161,-37.741,-46.189,179.349,6.071,149.284
C06995=1149.165,-37.991,-46.178,179.346,6.071,149.285
C06996=1149.171,-38.241,-46.166,179.344,6.070,149.285
C06997=1149.176,-38.491,-46.154,179.342,6.069,149.286
C06998=1149.181,-38.740,-46.143,179.339,6.069,149.286
C06999=1149.187,-38.989,-46.131,179.337,6.068,149.287
C07000=1149.192,-39.239,-46.120,179.335,6.067,149.287
C07001=1149.197,-39.489,-46.108,179.332,6.067,149.288
C07002=1149.202,-39.739,-46.096,179.330,6.066,149.289
C07003=1149.207,-39.989,-46.085,179.328,6.066,149.289
C07004=1149.213,-40.238,-46.074,179.325,6.066,149.290
C07005=1149.218,-40.488,-46.063,179.323,6.065,149.290
C07006=1149.224,-40.738,-46.051,179.321,6.065,149.291
C07007=1149.228,-40.988,-46.040,179.318,6.064,149.291
C07008=1149.234,-41.237,-46.028,179.316,6.063,149.292
C07009=1149.239,-41.486,-46.017,179.314,6.063,149.293
C07010=1149.244,-41.736,-46.005,179.311,6.062,149.293
C07011=1149.249,-41.986,-45.994,179.309,6.061,149.294
C07012=1149.255,-42.236,-45.982,179.307,6.061,149.294
C07013=1149.260,-42.485,-45.971,179.304,6.060,149.295
C07014=1149.265,-42.735,-45.959,179.302,6.059,149.295
C07015=1149.270,-42.984,-45.948,179.300,6.059,149.296
C07016=1149.276,-43.235,-45.937,179.297,6.059,149.297
C07017=1149.280,-43.485,-45.925,179.295,6.058,149.297
C07018=1149.286,-43.734,-45.914,179.293,6.058,149.298
C07019=1149.291,-43.983,-45.902,179.290,6.057,149.298
C07020=1149.297,-44.233,-45.891,179.288,6.057,149.299
C07021=1149.301,-44.483,-45.879,179.286,6.056,149.299
C07022=1149.307,-44.732,-45.868,179.283,6.055,149.300
C07023=1149.312,-44.982,-45.857,179.281,6.055,149.301
C07024=1149.317,-45.232,-45.846,179.278,6.054,149.301
C07025=1149.323,-45.481,-45.834,179.276,6.054,149.302
C07026=1149.328,-45.731,-45.823,179.274,6.054,149.302
C07027=1149.333,-45.981,-45.811,179.272,6.053,149.303
C07028=1149.338,-46.231,-45.801,179.269,6.052,149.303
C07029=1149.344,-46.480,-45.789,179.267,6.052,149.304
C07030=1149.349,-46.730,-45.778,179.265,6.051,149.305
C07031=1149.354,-46.980,-45.766,179.262,6.050,149.305
C07032=1149.360,-47.229,-45.756,179.260,6.050,149.306
C07033=1149.365,-47.479,-45.744,179.258,6.050,149.306
C07034=1149.370,-47.729,-45.732,179.256,6.049,149.307
C07035=1149.375,-47.978,-45.722,179.253,6.049,149.307
C07036=1149.380,-48.228,-45.711,179.251,6.048,149.308
C07037=1149.386,-48.478,-45.699,179.249,6.047,149.308
C07038=1149.390,-48.728,-45.688,179.246,6.047,149.309
C07039=1149.396,-48.977,-45.678,179.244,6.046,149.310
C07040=1149.401,-49.227,-45.666,179.241,6.046,149.310
C07041=1149.406,-49.477,-45.654,179.240,6.046,149.311
C07042=1149.411,-49.726,-45.644,179.237,6.045,149.311
C07043=1149.417,-49.976,-45.632,179.235,6.044,149.312
C07044=1149.423,-50.247,-45.620,179.232,6.044,149.313
C07045=1149.428,-50.517,-45.609,179.230,6.043,149.313
C07046=1149.434,-50.788,-45.597,179.227,6.043,149.314
C07047=1149.440,-51.059,-45.585,179.225,6.042,149.314
C07048=1149.445,-51.308,-45.573,179.223,6.042,149.315
C07049=1149.450,-51.558,-45.561,179.220,6.041,149.315
C07050=1149.456,-51.808,-45.551,179.218,6.041,149.316
C07051=1149.460,-52.057,-45.540,179.215,6.040,149.317
C07052=1149.466,-52.308,-45.529,179.213,6.039,149.317
C07053=1149.471,-52.557,-45.518,179.211,6.039,149.318
C07054=1149.476,-52.806,-45.507,179.209,6.039,149.318
C07055=1149.482,-53.056,-45.496,179.206,6.038,149.319
C07056=1149.487,-53.306,-45.485,179.204,6.037,149.319
C07057=1149.492,-53.556,-45.474,179.202,6.037,149.320
C07058=1149.498,-53.805,-45.463,179.199,6.036,149.321
C07059=1149.503,-54.055,-45.452,179.198,6.036,149.321
C07060=1149.509,-54.305,-45.441,179.195,6.036,149.322
C07061=1149.514,-54.555,-45.430,179.193,6.035,149.322
C07062=1149.518,-54.804,-45.419,179.191,6.034,149.323
C07063=1149.524,-55.053,-45.408,179.188,6.034,149.323
C07064=1149.529,-55.304,-45.397,179.186,6.033,149.324
C07065=1149.535,-55.553,-45.386,179.184,6.033,149.324
C07066=1149.540,-55.803,-45.375,179.182,6.033,149.325
C07067=1149.544,-56.053,-45.364,179.179,6.032,149.326
C07068=1149.550,-56.302,-45.354,179.177,6.032,149.326
C07069=1149.555,-56.552,-45.343,179.175,6.031,149.327
C07070=1149.561,-56.802,-45.332,179.172,6.030,149.327
C07071=1149.566,-57.052,-45.321,179.170,6.030,149.328
C07072=1149.571,-57.301,-45.310,179.168,6.030,149.328
C07073=1149.576,-57.551,-45.300,179.165,6.029,149.329
C07074=1149.581,-57.801,-45.289,179.163,6.028,149.330
C07075=1149.586,-58.050,-45.278,179.161,6.028,149.330
C07076=1149.592,-58.300,-45.266,179.158,6.027,149.331
C07077=1149.597,-58.550,-45.256,179.157,6.027,149.331
C07078=1149.602,-58.800,-45.246,179.155,6.026,149.332
C07079=1149.608,-59.049,-45.235,179.152,6.026,149.332
C07080=1149.613,-59.299,-45.224,179.150,6.025,149.333
C07081=1149.618,-59.548,-45.213,179.147,6.025,149.334
C07082=1149.623,-59.798,-45.203,179.145,6.025,149.334
C07083=1149.629,-60.048,-45.192,179.143,6.024,149.335
C07084=1149.634,-60.298,-45.181,179.141,6.024,149.335
C07085=1149.640,-60.547,-45.170,179.138,6.023,149.336
C07086=1149.645,-60.798,-45.160,179.136,6.023,149.337
C07087=1149.650,-61.047,-45.149,179.134,6.022,149.337
C07088=1149.655,-61.297,-45.138,179.132,6.022,149.337
C07089=1149.661,-61.546,-45.128,179.129,6.021,149.338
C07090=1149.665,-61.796,-45.117,179.127,6.021,149.339
C07091=1149.671,-62.045,-45.107,179.125,6.020,149.339
C07092=1149.676,-62.296,-45.096,179.122,6.019,149.340
C07093=1149.681,-62.545,-45.085,179.121,6.019,149.340
C07094=1149.686,-62.795,-45.074,179.118,6.019,149.341
C07095=1149.692,-63.045,-45.064,179.116,6.018,149.342
C07096=1149.697,-63.295,-45.053,179.114,6.018,149.342
C07097=1149.703,-63.544,-45.042,179.111,6.017,149.343
C07098=1149.708,-63.794,-45.032,179.109,6.017,149.343
C07099=1149.713,-64.044,-45.021,179.107,6.016,149.344
C07100=1149.718,-64.293,-45.010,179.104,6.016,149.344
C07101=1149.724,-64.543,-45.000,179.102,6.015,149.345
C07102=1149.729,-64.792,-44.990,179.101,6.015,149.345
C07103=1149.734,-65.043,-44.979,179.098,6.015,149.346
C07104=1149.740,-65.292,-44.969,179.096,6.014,149.347
C07105=1149.745,-65.542,-44.958,179.093,6.014,149.347
C07106=1149.750,-65.791,-44.947,179.091,6.013,149.348
C07107=1149.755,-66.042,-44.937,179.089,6.013,149.348
C07108=1149.761,-66.291,-44.927,179.087,6.013,149.349
C07109=1149.766,-66.541,-44.916,179.085,6.012,149.349
C07110=1149.771,-66.790,-44.905,179.082,6.011,149.350
C07111=1149.777,-67.040,-44.895,179.080,6.011,149.351
C07112=1149.782,-67.290,-44.884,179.078,6.011,149.351
C07113=1149.787,-67.540,-44.874,179.076,6.010,149.352
C07114=1149.792,-67.790,-44.864,179.073,6.009,149.352
C07115=1149.798,-68.039,-44.853,179.071,6.009,149.353
C07116=1149.803,-68.289,-44.843,179.069,6.009,149.353
C07117=1149.807,-68.538,-44.832,179.067,6.008,149.354
C07118=1149.813,-68.788,-44.822,179.065,6.008,149.354
C07119=1149.818,-69.038,-44.812,179.062,6.007,149.355
C07120=1149.824,-69.288,-44.801,179.060,6.007,149.356
C07121=1149.829,-69.537,-44.791,179.058,6.006,149.356
C07122=1149.834,-69.787,-44.781,179.055,6.006,149.357
C07123=1149.840,-70.037,-44.770,179.053,6.005,149.357
C07124=1149.845,-70.287,-44.760,179.052,6.005,149.358
C07125=1149.850,-70.537,-44.750,179.049,6.005,149.358
C07126=1149.856,-70.786,-44.739,179.047,6.004,149.359
C07127=1149.862,-71.036,-44.729,179.045,6.003,149.359
C07128=1149.867,-71.286,-44.719,179.043,6.004,149.360
C07129=1149.871,-71.535,-44.709,179.040,6.003,149.361
C07130=1149.876,-71.786,-44.698,179.038,6.002,149.361
C07131=1149.882,-72.035,-44.688,179.035,6.002,149.362
C07132=1149.888,-72.285,-44.678,179.034,6.002,149.362
C07133=1149.893,-72.535,-44.668,179.032,6.001,149.363
C07134=1149.898,-72.784,-44.657,179.029,6.001,149.363
C07135=1149.904,-73.034,-44.647,179.027,6.000,149.364
C07136=1149.909,-73.284,-44.637,179.025,6.000,149.364
C07137=1149.914,-73.533,-44.627,179.023,6.000,149.365
C07138=1149.919,-73.783,-44.617,179.020,5.999,149.366
C07139=1149.925,-74.033,-44.606,179.018,5.998,149.366
C07140=1149.930,-74.283,-44.596,179.016,5.998,149.367
C07141=1149.935,-74.532,-44.586,179.014,5.998,149.367
C07142=1149.941,-74.782,-44.575,179.011,5.997,149.368
C07143=1149.945,-75.032,-44.566,179.009,5.996,149.368
C07144=1149.951,-75.281,-44.555,179.007,5.997,149.369
C07145=1149.956,-75.531,-44.545,179.005,5.996,149.370
C07146=1149.961,-75.781,-44.535,179.003,5.995,149.370
C07147=1149.967,-76.031,-44.524,179.000,5.995,149.371
C07148=1149.973,-76.301,-44.514,178.998,5.995,149.371
C07149=1149.979,-76.574,-44.503,178.996,5.994,149.372
C07150=1149.984,-76.845,-44.492,178.993,5.994,149.373
C07151=1149.989,-77.116,-44.481,178.991,5.993,149.373
C07152=1149.995,-77.366,-44.471,178.989,5.993,149.374
C07153=1150.001,-77.615,-44.461,178.987,5.993,149.374
C07154=1150.006,-77.865,-44.450,178.985,5.992,149.375
C07155=1150.012,-78.116,-44.441,178.982,5.992,149.375
C07156=1150.016,-78.365,-44.431,178.980,5.991,149.376
C07157=1150.022,-78.614,-44.421,178.978,5.991,149.376
C07158=1150.028,-78.864,-44.411,178.976,5.990,149.377
C07159=1150.033,-79.114,-44.400,178.973,5.990,149.378
C07160=1150.037,-79.363,-44.390,178.972,5.990,149.378
C07161=1150.043,-79.614,-44.381,178.969,5.989,149.379
C07162=1150.049,-79.863,-44.371,178.967,5.989,149.379
C07163=1150.053,-80.113,-44.361,178.965,5.988,149.380
C07164=1150.059,-80.363,-44.350,178.963,5.988,149.380
C07165=1150.064,-80.612,-44.340,178.961,5.987,149.381
C07166=1150.070,-80.862,-44.331,178.958,5.987,149.381
C07167=1150.075,-81.112,-44.321,178.957,5.987,149.382
C07168=1150.080,-81.362,-44.311,178.954,5.986,149.383
C07169=1150.086,-81.611,-44.300,178.952,5.986,149.383
C07170=1150.091,-81.861,-44.291,178.950,5.985,149.384
C07171=1150.097,-82.111,-44.281,178.948,5.985,149.384
C07172=1150.102,-82.360,-44.271,178.945,5.984,149.385
C07173=1150.106,-82.610,-44.261,178.943,5.984,149.385
C07174=1150.112,-82.860,-44.252,178.941,5.984,149.386
C07175=1150.117,-83.110,-44.242,178.939,5.983,149.386
C07176=1150.123,-83.359,-44.232,178.937,5.983,149.387
C07177=1150.129,-83.609,-44.222,178.935,5.983,149.387
C07178=1150.133,-83.859,-44.212,178.933,5.982,149.388
C07179=1150.139,-84.109,-44.202,178.930,5.981,149.389
C07180=1150.144,-84.359,-44.193,178.928,5.981,149.389
C07181=1150.149,-84.608,-44.183,178.926,5.981,149.390
C07182=1150.155,-84.858,-44.173,178.924,5.980,149.390
C07183=1150.159,-85.108,-44.163,178.922,5.980,149.391
C07184=1150.165,-85.358,-44.153,178.920,5.980,149.391
C07185=1150.171,-85.607,-44.143,178.917,5.979,149.392
C07186=1150.176,-85.857,-44.134,178.915,5.978,149.392
C07187=1150.181,-86.107,-44.124,178.914,5.978,149.393
C07188=1150.186,-86.356,-44.114,178.911,5.978,149.394
C07189=1150.192,-86.606,-44.105,178.909,5.977,149.394
C07190=1150.197,-86.856,-44.094,178.907,5.977,149.395
C07191=1150.202,-87.106,-44.085,178.905,5.977,149.395
C07192=1150.208,-87.356,-44.075,178.902,5.976,149.396
C07193=1150.213,-87.605,-44.066,178.901,5.976,149.396
C07194=1150.219,-87.855,-44.056,178.898,5.976,149.397
C07195=1150.224,-88.104,-44.046,178.896,5.975,149.397
C07196=1150.230,-88.355,-44.037,178.894,5.975,149.398
C07197=1150.234,-88.604,-44.027,178.892,5.974,149.398
C07198=1150.240,-88.855,-44.017,178.889,5.974,149.399
C07199=1150.245,-89.104,-44.008,178.888,5.974,149.400
C07200=1150.250,-89.353,-43.998,178.886,5.973,149.400
C07201=1150.255,-89.603,-43.989,178.883,5.972,149.401
C07202=1150.261,-89.853,-43.979,178.881,5.973,149.401
C07203=1150.266,-90.103,-43.970,178.879,5.972,149.402
C07204=1150.272,-90.352,-43.959,178.877,5.971,149.402
C07205=1150.277,-90.602,-43.951,178.875,5.972,149.403
C07206=1150.282,-90.852,-43.940,178.873,5.971,149.403
C07207=1150.287,-91.102,-43.931,178.870,5.970,149.404
C07208=1150.293,-91.352,-43.921,178.869,5.970,149.404
C07209=1150.298,-91.602,-43.912,178.866,5.970,149.405
C07210=1150.303,-91.851,-43.902,178.864,5.969,149.406
C07211=1150.309,-92.101,-43.893,178.862,5.969,149.406
C07212=1150.314,-92.351,-43.883,178.860,5.969,149.407
C07213=1150.319,-92.600,-43.874,178.858,5.968,149.407
C07214=1150.325,-92.851,-43.864,178.856,5.968,149.408
C07215=1150.330,-93.100,-43.855,178.854,5.967,149.408
C07216=1150.336,-93.350,-43.845,178.851,5.967,149.409
C07217=1150.341,-93.599,-43.836,178.850,5.967,149.409
C07218=1150.346,-93.849,-43.827,178.847,5.966,149.410
C07219=1150.352,-94.099,-43.817,178.846,5.966,149.410
C07220=1150.357,-94.348,-43.808,178.843,5.966,149.411
C07221=1150.363,-94.599,-43.798,178.841,5.965,149.412
C07222=1150.368,-94.848,-43.788,178.839,5.965,149.412
C07223=1150.373,-95.098,-43.779,178.837,5.964,149.413
C07224=1150.378,-95.349,-43.770,178.834,5.964,149.413
C07225=1150.383,-95.598,-43.760,178.833,5.964,149.414
C07226=1150.389,-95.848,-43.751,178.831,5.963,149.414
C07227=1150.394,-96.097,-43.741,178.828,5.962,149.415
C07228=1150.400,-96.347,-43.731,178.826,5.963,149.415
C07229=1150.405,-96.597,-43.723,178.824,5.962,149.416
C07230=1150.410,-96.846,-43.713,178.823,5.962,149.416
C07231=1150.415,-97.097,-43.703,178.820,5.961,149.417
C07232=1150.421,-97.346,-43.695,178.818,5.961,149.418
C07233=1150.426,-97.596,-43.686,178.816,5.961,149.418
C07234=1150.431,-97.846,-43.675,178.814,5.960,149.419
C07235=1150.437,-98.096,-43.667,178.812,5.960,149.419
C07236=1150.442,-98.346,-43.657,178.810,5.960,149.420
C07237=1150.447,-98.595,-43.647,178.807,5.959,149.420
C07238=1150.452,-98.845,-43.639,178.806,5.959,149.421
C07239=1150.459,-99.094,-43.629,178.804,5.958,149.421
C07240=1150.464,-99.344,-43.620,178.801,5.958,149.422
C07241=1150.469,-99.593,-43.611,178.799,5.958,149.422
C07242=1150.475,-99.844,-43.601,178.797,5.957,149.423
C07243=1150.480,-100.093,-43.593,178.795,5.957,149.423
C07244=1150.485,-100.343,-43.583,178.793,5.957,149.424
C07245=1150.491,-100.593,-43.573,178.791,5.956,149.425
C07246=1150.496,-100.843,-43.565,178.789,5.956,149.425
C07247=1150.501,-101.093,-43.556,178.787,5.956,149.426
C07248=1150.506,-101.342,-43.547,178.785,5.955,149.426
C07249=1150.512,-101.592,-43.537,178.783,5.955,149.427
C07250=1150.517,-101.842,-43.528,178.780,5.954,149.427
C07251=1150.522,-102.092,-43.519,178.779,5.955,149.428
C07252=1150.528,-102.364,-43.508,178.776,5.954,149.428
C07253=1150.534,-102.636,-43.498,178.774,5.953,149.429
C07254=1150.540,-102.908,-43.489,178.772,5.953,149.429
C07255=1150.546,-103.180,-43.478,178.770,5.953,149.430
C07256=1150.551,-103.429,-43.469,178.767,5.952,149.431
C07257=1150.556,-103.679,-43.460,178.765,5.952,149.431
C07258=1150.561,-103.929,-43.452,178.764,5.952,149.432
C07259=1150.567,-104.179,-43.442,178.761,5.951,149.432
C07260=1150.572,-104.429,-43.433,178.759,5.951,149.433
C07261=1150.578,-104.679,-43.424,178.757,5.950,149.433
C07262=1150.582,-104.928,-43.415,178.755,5.950,149.434
C07263=1150.588,-105.178,-43.405,178.753,5.950,149.434
C07264=1150.594,-105.428,-43.396,178.751,5.949,149.435
C07265=1150.599,-105.677,-43.388,178.749,5.949,149.435
C07266=1150.604,-105.927,-43.379,178.747,5.949,149.436
C07267=1150.610,-106.177,-43.370,178.745,5.948,149.436
C07268=1150.616,-106.427,-43.360,178.743,5.948,149.437
C07269=1150.621,-106.677,-43.352,178.740,5.948,149.438
C07270=1150.626,-106.927,-43.343,178.739,5.948,149.438
C07271=1150.631,-107.177,-43.334,178.737,5.947,149.439
C07272=1150.636,-107.427,-43.325,178.735,5.947,149.439
C07273=1150.641,-107.676,-43.315,178.732,5.947,149.440
C07274=1150.648,-107.925,-43.306,178.730,5.946,149.440
C07275=1150.653,-108.175,-43.297,178.729,5.946,149.441
C07276=1150.658,-108.425,-43.288,178.726,5.945,149.441
C07277=1150.663,-108.675,-43.279,178.725,5.945,149.442
C07278=1150.668,-108.925,-43.271,178.722,5.945,149.442
C07279=1150.673,-109.175,-43.262,178.721,5.945,149.443
C07280=1150.679,-109.425,-43.252,178.718,5.944,149.443
C07281=1150.685,-109.674,-43.244,178.716,5.943,149.444
C07282=1150.690,-109.924,-43.235,178.715,5.943,149.444
C07283=1150.695,-110.174,-43.226,178.712,5.943,149.445
C07284=1150.701,-110.423,-43.217,178.710,5.943,149.446
C07285=1150.706,-110.673,-43.208,178.708,5.942,149.446
C07286=1150.711,-110.923,-43.199,178.707,5.942,149.447
C07287=1150.717,-111.172,-43.191,178.704,5.941,149.447
C07288=1150.722,-111.422,-43.182,178.702,5.941,149.448
C07289=1150.728,-111.673,-43.173,178.700,5.941,149.448
C07290=1150.733,-111.923,-43.164,178.698,5.940,149.449
C07291=1150.738,-112.173,-43.155,178.696,5.940,149.449
C07292=1150.744,-112.422,-43.147,178.694,5.940,149.450
C07293=1150.749,-112.672,-43.138,178.692,5.940,149.450
C07294=1150.755,-112.921,-43.129,178.690,5.939,149.451
C07295=1150.760,-113.171,-43.120,178.688,5.939,149.451
C07296=1150.765,-113.421,-43.111,178.686,5.939,149.452
C07297=1150.771,-113.670,-43.102,178.684,5.938,149.452
C07298=1150.776,-113.920,-43.094,178.682,5.938,149.453
C07299=1150.781,-114.170,-43.085,178.680,5.937,149.453
C07300=1150.786,-114.421,-43.077,178.678,5.938,149.454
C07301=1150.792,-114.670,-43.068,178.676,5.937,149.455
C07302=1150.797,-114.920,-43.059,178.674,5.937,149.455
C07303=1150.803,-115.169,-43.050,178.672,5.936,149.456
C07304=1150.808,-115.420,-43.041,178.670,5.935,149.456
C07305=1150.814,-115.669,-43.032,178.668,5.935,149.456
C07306=1150.819,-115.919,-43.023,178.666,5.935,149.457
C07307=1150.825,-116.169,-43.015,178.664,5.935,149.458
C07308=1150.830,-116.419,-43.006,178.662,5.934,149.458
C07309=1150.835,-116.669,-42.997,178.660,5.934,149.459
C07310=1150.841,-116.918,-42.989,178.658,5.934,149.459
